//--------------------------------------------------------------------------------
// Stan maszyny naciśnieciu estopa 	
	E_Station.eAborting:                 	// Stan bezpiecznego zatrzymywania (po EStopie)
		bGate1:= FALSE;
		bGate2:= FALSE;
	
		ACT_ResetCommands();

		eState 						:=  E_Station.eAborted;  
		eRunningState				:=	E_CapFeederState.eReady;
		
//--------------------------------------------------------------------------------
// Stan masyzny po wykryciu błędu			
	E_Station.eError:                 	 	// Stan błędu 	
		
		ACT_ResetCommands();
		
		IF bReset THEN
			eState 				:= E_Station.eResetting;
			bError := FALSE;
		END_IF
		
//--------------------------------------------------------------------------------
// Stan masyzny po wykryciu błędu
	E_Station.eResetting:					// Stan resetowania bledu (po Errorze)
			CASE udiErrorID-udiStationIndex OF
		
				//Error 8 - Błąd falownika
				266:
					fbInverter.bReset	:= TRUE;
					bError 				:= FALSE;
				ELSE
					bError := FALSE;	
			END_CASE		
		
		IF NOT bError AND fbInverter.eState = E_Station.eReady THEN
			fbInverter.bReset	:= FALSE;	
			
			udiErrorID 			:=	0;
			sErrorDescription 	:=	'';
			eState 				:=	E_Station.ePreparingToReady;
			eRunningState		:=	E_CapFeederState.eReady;
		ELSE
			eState 				:=	E_Station.eError;
		END_IF
    
//--------------------------------------------------------------------------------
// Stan ruchoow manualnych
	E_Station.eManualMovement:     			// Stan ruchów manualnych  
   
		ACT_ManualMovements();
		//Wyjście z trybu serwisowego
		IF NOT bManualMovement THEN
			
			bHeightMotorUp				:=	FALSE;
			bHeightMotorDown			:=	FALSE;
			
			eState:=E_Station.eReady;
		END_IF
		

//--------------------------------------------------------------------------------
// Stan rozpoczecia bazowania
	E_Station.eHoming:						// Stan bazowania 
		
		ACT_Homing();
		IF NOT bHoming AND NOT bHeightSet THEN
			bHeightMotorDown					:=	FALSE;
			bHeightMotorUp						:=	FALSE;
		   eState								:=E_Station.ePreparingToReady;
		END_IF		
		
//--------------------------------------------------------------------------------
// Stan zakończenia bazowania
	E_Station.eHomingDone:                  // Stan wykonania bazowania 
	
		bHeightMotorDown					:=	FALSE;
		bHeightMotorUp						:=	FALSE;
		bHeightMotorEncoderCounterReset		:=	FALSE;
		bHomingDone							:=	TRUE;
		IF NOT bHoming AND NOT bHeightSet THEN
		   eState:=E_Station.eReady;
		END_IF
		
//--------------------------------------------------------------------------------
// Stan przygotowania do gotowości
	E_Station.ePreparingToReady:            // Stan przygotowywania do gotowosci (zawsze przed Ready)  
		
		bGate1:= FALSE;
		bGate2:= FALSE;
	
		bSorterEngine:=FALSE;
		bSorterAir:=FALSE;
		
		eRunningState:=E_CapFeederState.eReady;
		eState:=E_Station.eReady;	
		
//-------------------------------------------------------------------------------
// Stan przygotowania do wyłączenia maszyny
	E_Station.ePreparingToDisable:          // Stan przygotowywania do nieaktywnosci (po wyłączeniu Enable) 
		
		bGate1:= FALSE;
		bGate2:= FALSE;
	
		bSorterEngine:=FALSE;
		bSorterAir:=FALSE;
		bHeightMotorUp:= NOT tonHomingSensor.Q;
		bHeightMotorDown:=FALSE;	
		IF tonHeightNoChange.Q OR tonHeightNoChangeTime.Q THEN
			bHeightMotorUp			:=	FALSE;
			bHeightMotorDown		:=	FALSE;	
			eRunningState			:=	E_CapFeederState.eReady;		
			eState					:=	E_Station.eDisabled;
		END_IF	
			
//--------------------------------------------------------------------------------
// Stan gotowości
	E_Station.eReady:						// Stan gotowosci 
	
		IF bRun AND NOT bCycleDone AND NOT bCycleNotDone THEN
			eState 				:= E_Station.eStarting; 
		END_IF
		IF bHoming OR bHeightSet THEN
			bHomingDone							:=	FALSE;
			eState 								:= E_Station.eHoming; 
		END_IF
		IF bManualMovement THEN
			//Jeśli przejście w tryb ruchów manualnych przepisz wszystkie stany siłowników sterowanych przez moduł
			//aby zapobiec ewentualnym kolizjom po wejściu w tryb serwisowy
			
			bManualHeightMotorUp		:= bHeightMotorUp;
			bManualHeightMotorDown		:= bHeightMotorDown;
			
			eState 						:= E_Station.eManualMovement; 
		END_IF
		IF NOT bRun THEN
			bCycleDone 			:= FALSE;
			bCycleNotDone 		:= FALSE;			
		END_IF
		
//--------------------------------------------------------------------------------
// Stan zatrzymywania
	E_Station.eStopping:					// Stan zatrzymywania 
		
		bSorterAir 		:= 	TRUE;
		bSorterEngine 	:=	FALSE;
		IF tonStoppingTime.Q THEN
			ACT_ResetCommands();
			eRunningState							:= E_CapFeederState.eReady;
			eState									:= E_Station.eReady;
		END_IF

		
//--------------------------------------------------------------------------------
// Stan uruchomienia lini ( po eReady)
	E_Station.eStarting:                  	// Stan uruchamiania (po Ready)
		iValvesCycleCase		:=0;
		eState					 := E_Station.eRunning; 

//--------------------------------------------------------------------------------
// Stan wykonywania pracy
	E_Station.eRunning:               		// Stan wykonywania cyklu (po Startingu), w tym stanie osobny

		ACT_Running();
		IF NOT bRun THEN 					(*Przerywanie cyklu*)
			eState				:= E_Station.eStopping;
			//bCycleNotDone		:= TRUE;
		END_IF
		(*IF bCycleDone OR bCycleNotDone THEN (*Cykl zakończony*)
			eState 				 := E_Station.eReady;
		END_IF*)						
		
		
END_CASE
END_ACTION

ACTION ACT_ErrorHandling:
//OBSŁUGA BŁĘDÓW STACJI SPRAWDZANIA
//************LISTA BŁĘDÓW***************
bStateError:= (eState=E_Station.eError) OR (eState=E_Station.eResetting) OR bIgnoreError;

//************LISTA BŁĘDÓW***************

//Error 1 - podnośnik nie porusza się pomimo wysterowania 
tonErrorHeightChange(IN:=(bHeightMotorUp OR bHeightMotorDown) AND lrLastHeightMotorPositionCV=lrHeightMotorPositionCV, PT:=T#3S);
tonEmptySleeveError(IN:=NOT bFullSleeveSensor AND bRun, PT:=INT_TO_TIME(iTimeToEmptySleeveError)*1000); //Było 30, teraz jest z receptur
tonMaxHeightError(IN:=lrHeightMotorPositionSV>lrMaxHeight AND NOT bHomingNeeded AND eState=E_Station.eReady,PT:=T#30S);
tonMinHeightError(IN:=lrHeightMotorPositionSV<lrMinHeight AND NOT bHomingNeeded AND eState=E_Station.eReady,PT:=T#30S);
tonSorterEngineError(IN:= NOT bEngineOK AND bSorterEngine, PT:=T#3S);
tonInverterError(IN:=fbInverter.bError AND NOT bStateError, PT:=T#3S);

IF (bEnable OR (eState = E_Station.ePreparingToDisable)) AND NOT bIgnoreError THEN
	
	IF tonErrorHeightChange.Q THEN
		bError:=TRUE;
		udiErrorID:=261;
		//udiErrorID:= udiErrorID+udiStationIndex;
		sErrorDescription:='Blokada podnośnika lub brak zasilania - sprawdź czujnik lub odblokuj mechanicznie';	
		sErrorDescription2:='';
	END_IF
	
	
	IF tonSorterEngineError.Q THEN
		bError:=TRUE;
		udiErrorID:=262;
		//udiErrorID:= udiErrorID+udiStationIndex;
		sErrorDescription:='Bład zabezpieczenia silnika - sprawdź wyłącznik';	
		sErrorDescription2:='';	
	END_IF
	
	//Error 3 - Pusty rekaw sortera nasadek
	IF tonEmptySleeveError.Q THEN
		bError:=TRUE;
		udiErrorID:=263;
		//udiErrorID:= udiErrorID+udiStationIndex;
		sErrorDescription:='Pusty rękaw sortera - uzupełnij nasadki';
		sErrorDescription2:='';
	END_IF
	
	
	//Error 4 - Bład nastaw max
	IF tonMaxHeightError.Q  THEN
		bError:=TRUE;
		udiErrorID:=264;
		//udiErrorID:= udiErrorID+udiStationIndex;
		sErrorDescription:='Wartość zadana wysokości jest większa od maksymalnej - zmień ustawienia w recepturze';
		sErrorDescription2:=REAL_TO_STRING(LREAL_TO_INT(lrMaxHeight));
	END_IF
	
	//Error 5 - Bład nastaw min
	IF tonMinHeightError.Q THEN
		bError:=TRUE;
		udiErrorID:=265;
		//udiErrorID:= udiErrorID+udiStationIndex;
		sErrorDescription:='Wartość zadana wysokości jest mniejsza od minimalnej - zmień ustawienia w recepturze ';
		sErrorDescription2:=REAL_TO_STRING(LREAL_TO_INT(lrMinHeight));
	END_IF	
	
	//Error 6 - Bład falownika
	IF tonInverterError.Q THEN
		bError:=TRUE;
		udiErrorID:=266;
		//udiErrorID:= udiErrorID+udiStationIndex;
		sErrorDescription:='Błąd falownika';
		sErrorDescription2:='';
	END_IF		
	
	
	
ELSE
	bError	:=FALSE;
END_IF


//-----------------------------------------------------------------------
IF bError AND NOT bStateError THEN

	IF eLastState = eRunning THEN
		bCycleNotDone						:= TRUE;
	END_IF

	eState 									:= E_Station.eError;
END_IF


//------------------------------------------------------------------------

(*Wyświetlanie błedu na wyjściu*)
bError;

(*Przepisywanie nazwy stacji*)
sErrorStationName 							:= sStationName;

//Jezeli nie zbazowane to potrzebne bazowanie
IF NOT bHeightMotorEncoderHomed  THEN
	bHomingDone								:=	FALSE;
END_IF
END_ACTION

ACTION ACT_HeightMotor:
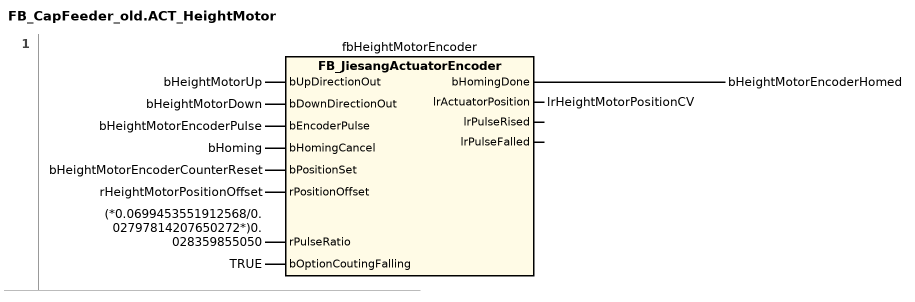
// NETWORK 1
fbHeightMotorEncoder(
    bUpDirectionOut := bHeightMotorUp,
    bDownDirectionOut := bHeightMotorDown,
    bEncoderPulse := bHeightMotorEncoderPulse,
    bHomingCancel := bHoming,
    bPositionSet := bHeightMotorEncoderCounterReset,
    rPositionOffset := rHeightMotorPositionOffset,
    rPulseRatio := (*0.0699453551912568/0.02797814207650272*)0.028359855050,
    bOptionCoutingFalling := TRUE,
    lrActuatorPosition => lrHeightMotorPositionCV); // FB_JiesangActuatorEncoder
bHeightMotorEncoderHomed := fbHeightMotorEncoder.bHomingDone;
END_ACTION

ACTION ACT_Homing:
//BAZOWANIE

tofHeightMotorDown(IN:=bHeightMotorDown, PT:=T#1S); //Zabezpieczenie przed zbyt szybkim przełączeniem pomiędzy Down a Up, bezpiecznieki sie palą
	
//Podnoszenie stacji do maksymalnej pozycji
IF NOT bHeightMotorEncoderHomed OR rtEncoderHomed.Q THEN
	bHeightMotorUp:=(*TRUE*) NOT tofHeightMotorDown.Q AND NOT tonHomingSensor.Q;
	bHeightMotorDown:=FALSE;
	IF tonHeightNoChange.Q OR tonHeightNoChangeTime.Q THEN
		bHeightMotorEncoderCounterReset:=TRUE;
		bHeightMotorUp:=FALSE;
    END_IF
	//Jesli enkoder zbazowany zakończ bazowanie	
	IF rtEncoderHomed.Q  THEN
		bHeightMotorUp:=FALSE;
		bHeightMotorDown:=FALSE;
		eState:=E_Station.eHomingDone;
	END_IF		
		
//Po podniesieniu stacji opuszczanie do ustalonej wysokości
ELSIF bHeightMotorEncoderHomed THEN
	bHeightMotorEncoderCounterReset:=FALSE;
	bHeightMotorUp:=lrHeightMotorPositionCV<=lrHeightMotorPositionSV;
	bHeightMotorDown:=lrHeightMotorPositionCV>=lrHeightMotorPositionSV;
	//Kiedy stacja osiągnie wysokość zadaną
	IF ABS(lrHeightMotorPositionCV-lrHeightMotorPositionSV)<0.5 OR tonLimitPosMaxReachedDelay.Q OR tonLimitPosMinReachedDelay.Q THEN
		bHeightMotorDown:=FALSE;
		bHeightMotorUp:=FALSE;
		eState:=E_Station.eHomingDone;
	END_IF			
END_IF
END_ACTION

ACTION ACT_Inverter:
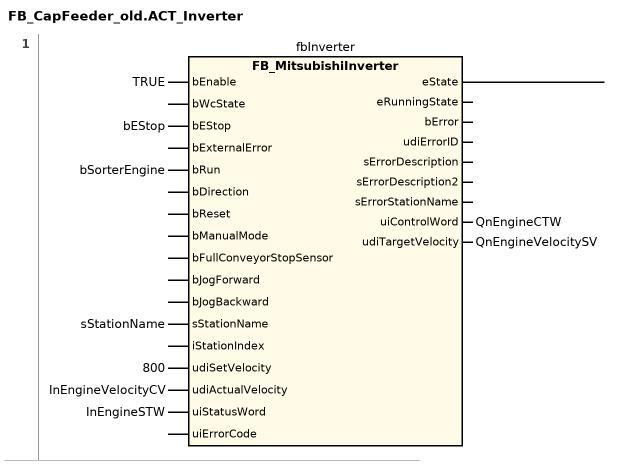
// NETWORK 1
fbInverter(
    bEnable := TRUE,
    bEStop := bEStop,
    bRun := bSorterEngine,
    sStationName := sStationName,
    udiSetVelocity := 800,
    udiActualVelocity := InEngineVelocityCV,
    uiStatusWord := InEngineSTW,
    uiControlWord => QnEngineCTW,
    udiTargetVelocity => QnEngineVelocitySV); // FB_MitsubishiInverter
END_ACTION

ACTION ACT_Limits:
IF iTimeToEmptySleeveError < 5 THEN
	iTimeToEmptySleeveError := 5;
END_IF
END_ACTION

ACTION ACT_ManualMovements:
//W trybie ruchów manualnych wykonuj ruchy za pomocą rozkazów manualnych
IF NOT bRun THEN
	
	bHeightMotorUp:=bManualHeightMotorUp;
	bHeightMotorDown:=bManualHeightMotorDown;
	bSorterEngine:=bManualSorterEngine;
	bSorterAir:=bManualSorterAir;
	
	bGate1:=bManualGate1; //Not dla tego, że defoltowy stan WYSUNIĘTY (true)
	bGate2:=bManualGate2; //Not dla tego, że defoltowy stan WYSUNIĘTY (true)

(*ELSE	//Kasuje zeby po cyklu nic sie nie poruszało

	bManualHeightMotorUp 	:= FALSE;
	bManualHeightMotorDown  := FALSE;
	bSorterEngine	:=FALSE;
	bSorterAir		:=FALSE;
*)	
END_IF


IF bHoming OR bHeightSet THEN
	eState:=E_Station.eHoming;
END_IF

IF bRun THEN	
	ACT_Running();
END_IF
//Zabezpieczenie przed kolizją stacji poprzez ruch podnośnika	
IF bHeightMotorDown AND lrHeightMotorPositionCV<=lrMinHeight AND NOT bHoming AND NOT bHeightSet THEN
	bHeightMotorDown:=FALSE;
END_IF	

IF bHeightMotorUp AND lrHeightMotorPositionCV>=lrMaxHeight AND NOT bHoming AND NOT bHeightSet THEN
	bHeightMotorUp:=FALSE;
END_IF
END_ACTION

ACTION ACT_ResetCommands:
//Reset komend ruchu 	


bHeightMotorUp				:=	FALSE;
bHeightMotorDown			:=	FALSE;
bSorterAir 		:= 	FALSE;
bSorterEngine 		:=	FALSE;
END_ACTION

ACTION ACT_Running:
//----------------------------------------------------------------------------------
// Obsługa podajnik zamknięc


(*CASE iValvesCycleCase OF
	0:
		bGate1:= FALSE;
		IF (tonGates1.Q) THEN
			iValvesCycleCase :=1;
		END_IF
	1:
		bGate1:= TRUE;
		IF (tonGates2.Q) THEN
			iValvesCycleCase :=2;
		END_IF	
	2:
		bGate2:= FALSE;
		IF (tonGates3.Q) THEN
			iValvesCycleCase :=3;
		END_IF
	3:
		bGate2:= TRUE;
		IF (tonGates4.Q) THEN
			iValvesCycleCase :=0;
		END_IF	
END_CASE*)

//rtOutSensor(CLK:=P08_CapSorter.IbCapSorterGateGateAfterSensor);
	
CASE iValvesCycleCase OF
	0:
		//IF (rtOutSensor.Q) THEN
		IF (NOT bSensorInPipe) THEN

			iValvesCycleCase:=1;
		END_IF
		;
	1:
		bGate1:= TRUE;
		IF (tonGates1.Q) THEN
			iValvesCycleCase :=2;
		END_IF
	2:
		bGate1:= FALSE;
		IF (tonGates2.Q) THEN
			iValvesCycleCase :=3;
		END_IF	
	3:
		bGate2:= TRUE;
		IF (tonGates3.Q) THEN
			iValvesCycleCase :=4;
		END_IF
	4:
		bGate2:= FALSE;
		IF (tonGates4.Q) THEN
			iValvesCycleCase :=0;
		END_IF	
END_CASE

CASE eRunningState OF
	
	//NIEGOTOWY
	E_CapFeederState.eDisabled:
		eRunningState:=E_CapFeederState.eReady;

	E_CapFeederState.eReady:
		iTryUnblockWheel		:=	0;
		bTryUnblockWheel		:= FALSE;	
		fbInverter.bDirection 	:= FALSE;
		IF bRun THEN
			eRunningState			:=E_CapFeederState.eSorting;
		END_IF
	
	
	E_CapFeederState.eSorting:
	
		bSorterEngine:=tonAirBeforeStart.Q;
		bSorterAir:=(	//Nie wiem co to za wymysły
						(aBufferedSensorValue[20](*tofCapFeederSorterCapSensor.Q*) OR NOT tonAirBeforeStart2.Q)(* AND bImpON*)AND NOT bBlowDelay
					)	OR	
					bTryUnblockWheel // Dmuchanie jeżeli jest obrót do tyłu
;
		//aBufferedSensorValue[20] - 20 to jest opóznenie (buferizacja signala czujnika w cyklach programy (3ms x 20 = 60 ms). Czas opóznenia 
		//możemy obliczyć od prędcosci falownika i prszykładni: mamy 51 gniazdk0, 800 rpm, przykladnia 1:40 => mamy 800/40=20rmp, /60 =>
		//0,33 obrota / sec => 0,33 obrota/sec * 51 dnazdko/obrot = 17 gniazdek/sek => 1/17 = 0,059sec/1gniazdko => opoznenie 60 ms
		//60ms/3ms(czas cyclu) => 20 cyclów
		
		(*Próba odblokowania koła*)
			iTryUnblockWheel := iTryUnblockWheel + 1;
			IF rtCapSorterSensor.Q THEN
				iTryUnblockWheel	:=	0;
			END_IF
			IF tonEngineBlocked.Q THEN
				bTryUnblockWheel := TRUE;
			END_IF	
			IF bTryUnblockWheel THEN
				fbInverter.bDirection := TRUE;
			END_IF
			IF tonTryUnblockWheel.Q THEN
				iTryUnblockWheel		:=	0;//dp
				bTryUnblockWheel		:= FALSE;
				fbInverter.bDirection 	:= FALSE;
			END_IF
		(* Koniec Próba odblokowania koła*)	
		
		IF tonSortingEngineOff.Q THEN 
			eRunningState 			:=E_CapFeederState.eSleeveFull;
		END_IF
	
	E_CapFeederState.eSleeveFull:
	
		bSorterEngine:=FALSE;
		bSorterAir:=NOT tonAirAfterStop.Q(* AND bImpON*);
		IF tonAirAfterStop.Q THEN
			IF tonSortingEngineOn.Q THEN
				eRunningState		:=E_CapFeederState.eSorting; 
			END_IF
		END_IF
	
	E_CapFeederState.eSleeveLowLevel:
	
			//Wlaczenie silnika i zaworu po czasie
		bSorterEngine:=TRUE;
		bSorterAir:=tofCapFeederSorterCapSensor.Q (*AND bImpON*);
		IF tonSortingEngineOff.Q THEN
			eRunningState		 	:=E_CapFeederState.eSorting;
		END_IF
	
END_CASE
END_ACTION

ACTION ACT_Signals:
(** Timery na potrzeby bazowania**)
rtEncoderHomed(CLK:=bHeightMotorEncoderHomed,Q=>);
tonHeightNoChange(IN:=((bHeightMotorUp OR bHeightMotorDown OR tonHomingSensor.Q) AND (lrLastHeightMotorPositionCV=lrHeightMotorPositionCV)), PT:=T#500MS); 
tonHomingSensor(IN:=(bHomingSensor), PT:=T#100MS);
//tonHeightNoChangeTime(IN:=(eState = E_Station.eHoming OR eState = E_Station.ePreparingToDisable) AND bHeightMotorUp, PT:=T#8S); 

tonLimitPosMinReachedDelay(IN:=(lrHeightMotorPositionCV<=lrMinHeight) AND eState=E_Station.eHoming,PT:=T#2S);
tonLimitPosMaxReachedDelay(IN:=(lrHeightMotorPositionCV>=lrMaxHeight) AND eState=E_Station.eHoming,PT:=T#2S);
	
(** Timery używane podczas pracy stacji**)
tonSortingEngineOff(IN:=((eRunningState=E_CapFeederState.eSorting OR eRunningState=E_CapFeederState.eSleeveLowLevel) AND bRun AND bFullSleeveSensor),PT:=INT_TO_TIME(iTimeDelayOff));
tonSortingEngineOn(IN:=((eRunningState=E_CapFeederState.eSorting OR eRunningState=E_CapFeederState.eSleeveFull) AND bRun AND NOT bFullSleeveSensor),PT:=INT_TO_TIME(iTimeDelayOn));
tonSleeveFullEngineOn(IN:=(eRunningState=E_CapFeederState.eSleeveFull AND bRun AND NOT bFullSleeveSensor),PT:=INT_TO_TIME(iTimeDelayOff));
rtCapSorterSensor(CLK:=bSorterCapSensor, Q=>);
tonEngineBlocked(IN:=iTryUnblockWheel > 1500 AND bSorterEngine AND NOT bTryUnblockWheel,PT:=T#1MS); //Zablokowany silnik
tonTryUnblockWheel(IN:=bTryUnblockWheel, PT:=T#1S900MS);
tofCapFeederSorterCapSensor(IN:=tonCapFeederSorterCapSensor.Q,PT:=T#10MS); //bylo 200
tonCapFeederSorterCapSensor(IN:=bSorterCapSensor,PT:=T#3mS);//było 3ms
tonAirBeforeStart(IN:=eRunningState=E_CapFeederState.eSorting, PT:=T#1S);
rtCapFeederSorterCapSensor(CLK:=tofCapFeederSorterCapSensor.Q,Q=>);

tonAirBeforeStart2(IN:=eRunningState=E_CapFeederState.eSorting, PT:=T#2S);
tonAirAfterStop(IN:=eRunningState=E_CapFeederState.eSleeveFull, PT:=T#2S);

//prszesunęcie wartosci czujnika po buforu opoznenia 

FOR i:=40 TO 1 BY -1 DO
	aBufferedSensorValue[i] := aBufferedSensorValue[i-1];
END_FOR
aBufferedSensorValue[0] := bSorterCapSensor;

IF rtCapFeederSorterCapSensor.Q THEN
	bBlowDelay := TRUE;
	
END_IF
tonbBlowDelay(IN:=bBlowDelay,PT:=T#35MS);
IF tonbBlowDelay.Q THEN
	bBlowDelay:= FALSE;
END_IF
TimerOn (IN := NOT bImpOn, PT := T#10MS);
IF TimerOn.Q THEN
	bImpOn := TRUE;
END_IF
TimerOff (IN := bImpOn, PT := T#10MS);
IF TimerOff.Q THEN
	bImpON := FALSE;
END_IF

//Czasówki pneumatiki
//tonGates1(IN:= (iValvesCycleCase = 0 AND (eState = E_Station.eRunning OR eState = E_Station.eManualMovement)), PT:=T#300MS);//150//300
//tonGates2(IN:= (iValvesCycleCase = 1 AND (eState = E_Station.eRunning OR eState = E_Station.eManualMovement)), PT:=T#200MS);//500//300
//tonGates3(IN:= (iValvesCycleCase = 2 AND (eState = E_Station.eRunning OR eState = E_Station.eManualMovement)), PT:=T#300MS);//150//300
//tonGates4(IN:= (iValvesCycleCase = 3 AND (eState = E_Station.eRunning OR eState = E_Station.eManualMovement)), PT:=T#200MS);//500//300

//Czasówki pneumatiki
tonGates1(IN:= (iValvesCycleCase = 1 AND (eState = E_Station.eRunning OR eState = E_Station.eManualMovement)), PT:=T#200MS);//150//300
tonGates2(IN:= (iValvesCycleCase = 2 AND (eState = E_Station.eRunning OR eState = E_Station.eManualMovement)), PT:=T#200MS);//500//300
tonGates3(IN:= (iValvesCycleCase = 3 AND (eState = E_Station.eRunning OR eState = E_Station.eManualMovement)), PT:=T#200MS);//150//300
tonGates4(IN:= (iValvesCycleCase = 4 AND (eState = E_Station.eRunning OR eState = E_Station.eManualMovement)), PT:=T#200MS);//500//300


(** Dodatkowy timer przy zatrzymywaniu**)
tonStoppingTime( IN:= eState= E_Station.eStopping, PT:=T#2S);
END_ACTION

ACTION ACT_Statistic:
//Statystyka do zliczania czasu cyklu 
rtrigCycleTimerRead(CLK:=eRunningState=E_CapFeederState.eSleeveFull OR eRunningState=E_CapFeederState.eSleeveLowLevel);

	IF rtrigCycleTimerRead.Q THEN
		tCycleTime:=tonCycleTimer.ET;
		
	END_IF
	
tonCycleTimer(IN:=eRunningState= E_CapFeederState.eSorting , PT:=T#1D);
END_ACTION

ACTION ACT_Status:

(*Zapisywanie ostatniego stanu*)
	IF eLastStateTemp<>eState THEN
		eLastState := eLastStateTemp;
	END_IF
	eLastStateTemp := eState;
	
	IF eLastRunningStateTemp<>eRunningState THEN
		eLastRunningState := eLastRunningStateTemp;
	END_IF
	eLastRunningStateTemp := eRunningState;
(*Koniec Zapisywanie ostatniego stanu*)
END_ACTION

ACTION ACT_Warnings:
//Usrawianie warningów

//Filtrowanie czujnika ultradźwiękowego
fbbLevelSensor	(bIN:=NOT bLevelSensor AND (eRunningState=E_CapFeederState.eSorting OR eRunningState=E_CapFeederState.eSleeveLowLevel OR eRunningState=E_CapFeederState.eSleeveFull) , tFilterTimeOn:= T#5S, tFilterTimeOff:=T#5S , bOUT=> );


IF fbbLevelSensor.bOUT THEN
		bWarning1						:=	TRUE;			
		udiWarningID					:=	1;
		sWarningDescription				:=	'Nieski poziom w sorterze nasadek';
ELSE
		bWarning1						:=	FALSE;			
		udiWarningID					:=	0;
		sWarningDescription				:=	'';
END_IF
END_ACTION

ACTION aStationID:
udiStationID	:=	udiStationIndex;
END_ACTION

END_FUNCTION_BLOCK

// ---- POUs/FB/FB_CatchStationEnkoder.TcPOU
(*
Nazwa:			FB_CatchStation
Opis:			Chwytak pod stacjami 
Wersja:			v1.1
Data:			2023-02-22
Autor:			TW,DP
Urzadzenia:		Silownik chwytania, podnośnik JIESANG
Konfiguracja:	
Zmiany:
20230222 - Zwieksozmny czas bledu 9
Info:
- dodano błędy od nastaw powyżej max i min (error 7 i 8)
- dodawno bHomingNeeded
- wylaczanie wyjść zmiana 2 wylaczanie wyjsc jak zniknie Enable
*)


FUNCTION_BLOCK FB_CatchStationEnkoder
VAR_INPUT
	bEnable: BOOL;						//Zezwolenie na pracę
	bEStop:BOOL;						//Stop Awaryjny włączony
	bRun:BOOL;							//Rozkaz łapania 
	bHoming:BOOL;						//Zezwolenie na wykonanie bazowania i pozycjonowania podajnika
	bHeightSet:BOOL;					//Ustaw wysokość
	bChangeover:BOOL;					//Ustawianie na zadaną wysokość do wymiany elementów formatowych
	bChangeOver2:BOOL;
	bIgnoreError:BOOL;					//Ignorowania błędów cyklu pracy
	bReset:BOOL;						//Reset błędu, jeśli w stanie "eError"
	nGripperScrewerPosition   	:LREAL; // Aktualna pozycja serwa od podnoszenia
	nSafetyScrewerPosition		:LREAL;	// zadana bezpieczna pozycja 
	bScrewerbError				:BOOL;  // Sygnał błędu od zakręcarki
	nPositionHeightSV:LREAL;			//Wysokość zadana na której ma znajdować się stacja
	bOpenedActuatorSensor:BOOL;			//Czujnik otwarcia siłownika łapania
	bClosedActuatorSensor:BOOL;			//Czujnik otwarcia siłownika łapania
	lrMaxHeight:LREAL;					//Maksymalna wysokość podnośnika chwytaka
	lrMinHeight:LREAL;					//Minimalna wysokość podnośnika chwytaka
	bManualMovement:BOOL;				//Zezwolenie na ruchy ręcznę
	bUnlockColision:BOOL:=FALSE;		//Odblokowywanie możliwośći kolizji
	bAlarmSVCVDiffHeightDisable:BOOL;	//Wyłączenie alarmu od rożnicy wysokości zadanej od aktualnej
	bNoLifter:BOOL;						//Podnośnik
	
	_HEIGHTMOTOR_ 				:BOOL;
	udiHeightMotorEncoderVal	:UDINT;		//Ilość impulsów z modułu enkoderowego
	bHeightEncoderSetValDone	:BOOL;		//Zerowanie enkodera wykonane
	bHeightMotorEncoderPulse 	:BOOL;			//Sygnał impulsów enkodera siłownika
	rHeightMotorPositionOffset 	:REAL;		//Wysokość bazowani podnośnika

	_ALARMINFO_ :BOOL;
	iStationIndex:UDINT;					//Numer stacji 
	sStationName:STRING;					//Nazwa stacji	

	
END_VAR
VAR_OUTPUT
	eState: E_Station;						//Stan ogólny bloku
	eRunningState: E_CatchStationState;		//Stan wewnętrzny
	bError: BOOL;							//Błąd stacji
	nErrorNr: UDINT;						//Nr błędu podajnika platynek
	sErrorDescription:STRING(200);				//Opis błędu
	sErrorDescription2: STRING(200);				//Opis błędu 2
	sErrorStationName:STRING;				//Nazwa stacji
	udiStationID: UDINT;				// Nr stacji

	bCatchActuator:BOOL;					//Sterownie siłownika łapania opakowania
	bHeightMotorUp:BOOL;					//Sterowanie silnikiem podnośnika  - RUCH W GÓRĘ
	bHeightMotorDown:BOOL;					//Sterowanie silnikiem podnośnika  - RUCH W DÓŁ
	udiHeightMotorEncoderSetVal	:UDINT;		
	bHeightEncoderSetVal	:BOOL;		//Zerowanie enkodera
	lrHeightMotorCV:LREAL;					//Aktualna pozycja podnośnika
	tCycleTime:TIME;
	bHomingDone:BOOL;						//Wymagane ponowne bazowanie (blad podczas bazowania lub stop awaryjny)
	bCycleDone:BOOL;
	bCycleNotDone:BOOL;
END_VAR
VAR
	tonHeightNoChange: TON; 			//Timer wykrycia braku ruchu siłownika zmiany wysokości stacji
	nLastPositionHeightCV: LREAL;		//Pozycja podnośnika w poprzednim cyklu programu
	tonErrorHeightChange: TON; 			//Timer błędu podnośnika
	// Czas zadziałania siłownika
	tonCatchingTime: TON;
	// Timer blokady otwierania chwytaka
	tonOpeningBlocked: TON;
	rtEncoderHomed:R_TRIG;
	tonCycleTimer:TON;
	rtrigCycleTimerRead:R_TRIG;
	
	tofMotorUpPermition: TOF;
	tofMotorDownPermition: TOF;
	tonLimitPosMinReachedDelay: TON;
	tonLimitPosMaxReachedDelay: TON;
	tonMaxHeight		: TON;
	tonMinHeight		: TON;
	tonSVCVDiffHeight	: TON;
	
	//Podnośnik Jiesang	
	fbHeightMotorEncoder: FB_JiesangActuatorEncoderModul;//FB_JiesangActuatorEncoder;	// Blok enkodera podnośnika chwytaka stabilizującego pod zakręcarką	
	bHeightMotorEncoderCounterReset:BOOL; 				//Sygnał resetu enkodera
	bHeightMotorEncoderHomed:BOOL;						//Informacja od enkodera że jest zbazowany

	eLastState: E_Station;							//Stan ogólny bloku
	eLastRunningState: E_CatchStationState;			//Stan podbloku
	eLastStateTemp: E_Station;						//Stan ogólny bloku
	eLastRunningStateTemp: E_CatchStationState;		//Stan podbloku
	bStateError: BOOL;

	tonStopping: TON;
	tofHeightMotorDown: TOF;
	iCaseChangeover: INT;
	tonChangeOverLimitPosMinReachedDelay: TON;
	tonChangeoverLimitPosMaxReachedDelay: TON;
END_VAR

VAR_IN_OUT
	bManualCatchActuator:BOOL;		//Ruch ręczny siłownikiem podajnika platynek
	bManualHeightMotorUp:BOOL;			//Ruch ręczny podnośnika stacji w górę
	bManualHeightMotorDown:BOOL;		//Ruch ręczny podnośnika stacji w dół
END_VAR

HeightMotor();
ErrorHandling();
Control();
Changeover();
Statistics();
aStationID();
(*Zapisywanie ostatniego stanu*)
IF eLastStateTemp<>eState THEN
	eLastState := eLastStateTemp;
END_IF
eLastStateTemp := eState;
IF eLastRunningStateTemp<>eRunningState THEN
	eLastRunningState := eLastRunningStateTemp;
END_IF
eLastRunningStateTemp := eRunningState;
(*Koniec Zapisywanie ostatniego stanu*)


nLastPositionHeightCV:=lrHeightMotorCV;

ACTION aStationID:
udiStationID	:=	iStationIndex;
END_ACTION

ACTION Changeover:
tonChangeOverLimitPosMinReachedDelay(IN:=(lrHeightMotorCV<=lrMinHeight) AND bChangeover,PT:=T#2S);
tonChangeoverLimitPosMaxReachedDelay(IN:=(lrHeightMotorCV>=lrMaxHeight) AND bChangeover,PT:=T#2S);


//Przeniesione do PreparingToDisabled
(*CASE iCaseChangeover OF
	
	0: //Włączenie ustawiania
		IF bChangeover THEN
			iCaseChangeover := iCaseChangeover + 10;
			bHeightMotorDown:=FALSE;
			bHeightMotorUp:=FALSE;
		END_IF
		
	10: //Ustawianie stacji na wysokość 
		IF bHeightMotorEncoderHomed THEN
			bHeightMotorEncoderCounterReset	:=	FALSE;
			bHeightMotorUp					:=	lrHeightMotorCV	<=	200;
			bHeightMotorDown				:=	lrHeightMotorCV	>=	200;
			//Kiedy stacja osiągnie wysokość zadaną
			IF ABS(lrHeightMotorCV-nPositionHeightSV)<2 OR tonChangeoverLimitPosMaxReachedDelay.Q OR tonChangeOverLimitPosMinReachedDelay.Q  THEN
				bHeightMotorDown			:=	FALSE;
				bHeightMotorUp				:=	FALSE;
				iCaseChangeover 			:=	iCaseChangeover + 10;
			END_IF			
		ELSE
			bHeightMotorDown		:=	FALSE;
			bHeightMotorUp			:=	FALSE;
			iCaseChangeover 		:=  0;
		END_IF	
		
	20: //Czekanie na wyłączenie przezbrajania i ustawienie na odpowiednią wysokość z receptury
			IF NOT bChangeover THEN
				iCaseChangeover := iCaseChangeover + 10;
			END_IF
	30: //Ustawianie stacji na wysokość z receptury
		IF bHeightMotorEncoderHomed THEN
			bHeightMotorEncoderCounterReset	:=	FALSE;
			bHeightMotorUp					:=	lrHeightMotorCV	<=	nPositionHeightSV;
			bHeightMotorDown				:=	lrHeightMotorCV	>=	nPositionHeightSV;
			//Kiedy stacja osiągnie wysokość zadaną
			IF ABS(lrHeightMotorCV-nPositionHeightSV)<2 OR tonChangeoverLimitPosMaxReachedDelay.Q OR tonChangeOverLimitPosMinReachedDelay.Q  THEN
				bHeightMotorDown			:=	FALSE;
				bHeightMotorUp				:=	FALSE;
				iCaseChangeover 			:=	iCaseChangeover + 10;
			END_IF			
		ELSE
			bHeightMotorDown		:=	FALSE;
			bHeightMotorUp			:=	FALSE;
			iCaseChangeover 		:=  0;
		END_IF
	40: //Ustawianie stacji na wysokość z receptury	
		iCaseChangeover 		:=  0;

END_CASE
*)
END_ACTION

ACTION Control:

	(** TIMERY**)
	rtEncoderHomed(CLK:=bHeightMotorEncoderHomed,Q=>);
	tonHeightNoChange(IN:=((bHeightMotorUp OR bHeightMotorDown) AND (nLastPositionHeightCV=lrHeightMotorCV)), PT:=T#1S); 
	tonLimitPosMinReachedDelay(IN:=(lrHeightMotorCV<=lrMinHeight) AND eState=E_Station.eHoming,PT:=T#2S);
	tonLimitPosMaxReachedDelay(IN:=(lrHeightMotorCV>=lrMaxHeight) AND eState=E_Station.eHoming,PT:=T#2S);
	tonStopping(IN:=eState=E_Station.eStopping,PT:=T#2S);
	tofMotorUpPermition(IN:=bHeightMotorDown,PT:=T#250MS);
	tofMotorDownPermition(IN:=bHeightMotorUp ,PT:=T#250MS);	
	(*****Wyłączenie enable*****)
	IF NOT bEnable OR bChangeover THEN //Lub przezbrajania
		IF eState <> E_Station.eDisabled AND eState <> E_Station.ePreparingToDisable AND nGripperScrewerPosition>nSafetyScrewerPosition AND NOT bScrewerbError THEN
				eState 				:= E_Station.ePreparingToDisable; 
		END_IF	
	END_IF

	(*****Estop*****)
	IF NOT bEstop  THEN	
		IF eState <> E_Station.eAborted AND eState <> E_Station.eAborting AND eState <> E_Station.eDisabled THEN
				eState 				:= E_Station.eAborting; 
		END_IF
	END_IF

	CASE eState OF
	/////////////////////////////	
		E_Station.eDisabled: 					// Stan nieaktywnosci (Stacja wyłączona) 

			IF bEnable THEN
				eState 				:= E_Station.ePreparingToReady; 
			END_IF 
			
    /////////////////////////////	    
		E_Station.eAborted: 					// Stan bezpiecznego zatrzymania (po Abortingu) 

			IF bEStop THEN
				eState 				:= E_Station.ePreparingToReady;
			END_IF
			
	/////////////////////////////	
		E_Station.eAborting:                 	// Stan bezpiecznego zatrzymywania (po EStopie)

			bHeightMotorUp				:=	FALSE;
			bHeightMotorDown			:=	FALSE;
			eState := E_Station.eAborted;  
			eRunningState:=E_CatchStationState.eDisabled;
			
	/////////////////////////////			
		E_Station.eError:                 	 	// Stan błędu 	

			iCaseChangeover 		:=	0;
			IF bReset THEN
				eState 				:=	E_Station.eResetting;
			END_IF
						
	/////////////////////////////
		E_Station.eResetting:					// Stan resetowania bledu (po Errorze)
	
			bError := FALSE;

			IF NOT bError THEN
				nErrorNr 			:=	0;
   				sErrorDescription 	:=	'';
				eState 				:=	E_Station.ePreparingToReady;
			ELSE
				eState 				:=	E_Station.eError;
			END_IF
        
	/////////////////////////////
		E_Station.eManualMovement:     			// Stan ruchów manualnych  

			ManualMovements();
			//Wyjście z trybu serwisowego
			IF NOT bManualMovement THEN
				bCatchActuator				:=	FALSE;
				bHeightMotorUp				:=	FALSE;
				bHeightMotorDown			:=	FALSE;
				bManualCatchActuator		:=	bCatchActuator;
				eState:=E_Station.eReady;
			END_IF

	/////////////////////////////
		E_Station.eHoming:						// Stan bazowania 
	IF (nGripperScrewerPosition>nSafetyScrewerPosition AND NOT bScrewerbError) OR bManualMovement THEN  // co to za bzdura
			Homing();
			IF NOT bHoming AND NOT bHeightSet THEN // co to za bzdura
			   eState:=E_Station.ePreparingToReady;
			   	bHeightMotorDown:=FALSE;
				bHeightMotorUp:=FALSE;
			END_IF		
	END_IF		
	/////////////////////////////
		E_Station.eHomingDone:                  // Stan wykonania bazowania 
	
			bHeightMotorDown					:=	FALSE;
			bHeightMotorUp						:=	FALSE;
			bHeightMotorEncoderCounterReset		:=	FALSE;
			bHomingDone							:=	TRUE;
			IF NOT bHoming AND NOT bHeightSet THEN
			   eState:=E_Station.eReady;
			END_IF
			
	/////////////////////////////
		E_Station.ePreparingToReady:            // Stan przygotowywania do gotowosci (zawsze przed Ready)  
	
			bCatchActuator	:=	FALSE;
			eRunningState	:=	E_CatchStationState.eReady;
			eState			:=	E_Station.eReady;	
			
	/////////////////////////////
		E_Station.ePreparingToDisable:          // Stan przygotowywania do nieaktywnosci (po wyłączeniu Enable) 
  
			bCatchActuator:=FALSE;
			IF NOT bChangeOver THEN //Normalne wyłączenie
				bHeightMotorUp:=TRUE;
				bHeightMotorDown:=FALSE;	
				IF tonHeightNoChange.Q THEN
					bHeightMotorUp:=FALSE;
					eState:=E_Station.eDisabled;
					eRunningState:=E_CatchStationState.eDisabled;
				END_IF	
			ELSE //Wyłączenie z przebrajaniem na pozycje 200
				IF bHeightMotorEncoderHomed THEN
					bHeightMotorEncoderCounterReset	:=	FALSE;
					bHeightMotorUp					:=	lrHeightMotorCV	<=	150 AND NOT tofMotorUpPermition.Q;
					bHeightMotorDown				:=	lrHeightMotorCV	>=	150 AND NOT tofMotorDownPermition.Q;
					//Kiedy stacja osiągnie wysokość zadaną
					IF ABS(lrHeightMotorCV-150)<2 OR tonChangeoverLimitPosMaxReachedDelay.Q OR tonChangeOverLimitPosMinReachedDelay.Q  THEN
						bHeightMotorDown			:=	FALSE;
						bHeightMotorUp				:=	FALSE;
						eState						:=	E_Station.eDisabled;
						eRunningState				:=	E_CatchStationState.eDisabled;
					END_IF			
				ELSE
					bHeightMotorDown				:=	FALSE;
					bHeightMotorUp					:=	FALSE;
					eState								:=E_Station.eDisabled;
					eRunningState					:=	E_CatchStationState.eDisabled;
				END_IF	
			END_IF
				
	/////////////////////////////
		E_Station.eReady:						// Stan gotowosci 

			IF bRun AND NOT bCycleDone AND NOT bCycleNotDone THEN
				eState 				:= E_Station.eStarting; 
			END_IF
			IF bHoming OR bHeightSet OR bChangeover THEN
				eState 				:= E_Station.eHoming; 
			END_IF
			IF bManualMovement THEN
				//Jeśli przejście w tryb ruchów manualnych przepisz wszystkie stany siłowników sterowanych przez moduł
				//aby zapobiec ewentualnym kolizjom po wejściu w tryb serwisowy
				bManualCatchActuator		:= bCatchActuator;
				bManualHeightMotorUp		:= bHeightMotorUp;
				bManualHeightMotorDown		:= bHeightMotorDown;
				
				eState 						:= E_Station.eManualMovement; 
				eRunningState 				:= E_CatchStationState.eReady;
 
			END_IF
			IF NOT bRun THEN
				bCycleDone 			:= FALSE;
				bCycleNotDone 		:= FALSE;			
			END_IF
			
	/////////////////////////////
		E_Station.eStopping:					// Stan zatrzymywania 
					
			Running();
			IF bOpenedActuatorSensor OR tonStopping.Q THEN //NEW
				eState						:=	E_Station.eReady;
				eRunningState 				:=	E_CatchStationState.eReady;
			END_IF
			
	/////////////////////////////
		E_Station.eStarting:                  	// Stan uruchamiania (po Ready)
				
			eState					 := E_Station.eRunning; 

	/////////////////////////////
		E_Station.eRunning:               		// Stan wykonywania cyklu (po Startingu), w tym stanie osobny

			Running();
			IF NOT bRun THEN 					(*Przerywanie cyklu*)
				eState				:= E_Station.eStopping;
				bCycleNotDone		:= TRUE;
			END_IF
			(*IF bCycleDone OR bCycleNotDone THEN (*Cykl zakończony*)
				eState 				 := E_Station.eReady;
			END_IF*)						
		ELSE
		
		
	/////////////////////////////		
	END_CASE
END_ACTION

ACTION ErrorHandling:
//OBSŁUGA BŁĘDÓW PODAJNIKA PLATYNEK

//************LISTA BŁĘDÓW***************
bStateError:= (eState=E_Station.eError) OR (eState=E_Station.eResetting) OR bIgnoreError;




IF bEnable THEN
	
	//Error 1 - Blokada otwarcia chwytaka
	tonOpeningBlocked(IN:=NOT bCatchActuator AND NOT bOpenedActuatorSensor, PT:=T#3S);
	
	IF tonOpeningBlocked.Q AND NOT bStateError THEN
		sErrorDescription:='Blokada otwarcia chwytaka - sprawdź czujnik';
		bHeightMotorUp:=FALSE;
		bError := TRUE;
		nErrorNr:=281;	
		//nErrorNr := nErrorNr+iStationIndex;
	END_IF
	
	//Error 2 - podnośnik nie porusza się pomimo wysterowania 
	tonErrorHeightChange(IN:=(bHeightMotorUp OR bHeightMotorDown) AND nLastPositionHeightCV=lrHeightMotorCV AND NOT bNoLifter, PT:=T#3S);
	
	IF tonErrorHeightChange.Q AND NOT bStateError THEN
		bHeightMotorUp:=FALSE;
		bHeightMotorDown:=FALSE;
		bError := TRUE;
		nErrorNr:=282;
		//nErrorNr := nErrorNr+iStationIndex;
		sErrorDescription:='Blokada podnośnika lub brak zasilania - sprawdź czujnik lub odblokuj mechanicznie';	
	END_IF
	
	
	//Error 3 - Bład nastaw max
	tonMaxHeight(IN:=nPositionHeightSV>lrMaxHeight+1 AND bHomingDone AND lrMaxHeight>0 AND eState=E_Station.eReady,PT:=T#30S);
	IF tonMaxHeight.Q AND NOT bStateError THEN
		bHeightMotorUp:=FALSE;
		bHeightMotorDown:=FALSE;
		bError := TRUE;
		nErrorNr:=283;
		//nErrorNr := nErrorNr+iStationIndex;
		sErrorDescription:='Wartość zadana wysokości jest większa od maksymalnej - zmień ustawienia w recepturze';
		sErrorDescription2:=REAL_TO_STRING(LREAL_TO_INT(lrMaxHeight));
	END_IF
	
	//Error 4 - Bład nastaw min
	tonMinHeight(IN:=nPositionHeightSV<lrMinHeight-1 AND bHomingDone AND lrMinHeight>0 AND eState=E_Station.eReady,PT:=T#30S);
	IF tonMinHeight.Q AND NOT bStateError THEN
		bHeightMotorUp:=FALSE;
		bHeightMotorDown:=FALSE;
		bError := TRUE;
		nErrorNr:=284;
		//nErrorNr := nErrorNr+iStationIndex;
		sErrorDescription:='Wartość zadana wysokości jest mniejsza od minimalnej - zmień ustawienia w recepturze ';
		sErrorDescription2:=REAL_TO_STRING(LREAL_TO_INT(lrMinHeight));
	END_IF
	
	//Error 5 - Bład zbyt dużej różnicy nastaw
	//tonSVCVDiffHeight(IN:=ABS(nPositionHeightSV-lrHeightMotorCV)>10 AND bHomingDone AND NOT bAlarmSVCVDiffHeightDisable AND eState=E_Station.eReady AND NOT bChangeOver2,PT:=T#5M);
	IF tonSVCVDiffHeight.Q AND NOT bStateError THEN
		bHeightMotorUp:=FALSE;
		bHeightMotorDown:=FALSE;
		bError := TRUE;
		nErrorNr:=285;
		//nErrorNr := nErrorNr+iStationIndex;
		sErrorDescription:='Wartość aktualna jest zbyt różna od zadanej - zmień ustawienia w recepturze lub ustaw stację';
		sErrorDescription2:=REAL_TO_STRING(LREAL_TO_INT(nPositionHeightSV));
		
	END_IF	
		
	
	
ELSE
	bError := FALSE;
END_IF

	
//******************PRZEJŚCIE DO eERROR*****************************

IF bError AND NOT bStateError THEN
	IF eLastState = eRunning THEN
		bCycleNotDone := TRUE;
	END_IF
	eState := E_Station.eError;
END_IF

//****************WYŚWIETLANIE STATUSU BLEDU***********************

(*Wyświetlanie błedu na wyjściu*)
bError;

(*Przepisywanie nazwy stacji*)
sErrorStationName := sStationName;


//Jezeli nie zbazowane to potrzebne bazowanie
IF NOT bHeightMotorEncoderHomed AND NOT bNoLifter  THEN
	bHomingDone:=FALSE;
END_IF
END_ACTION

ACTION HeightMotor:
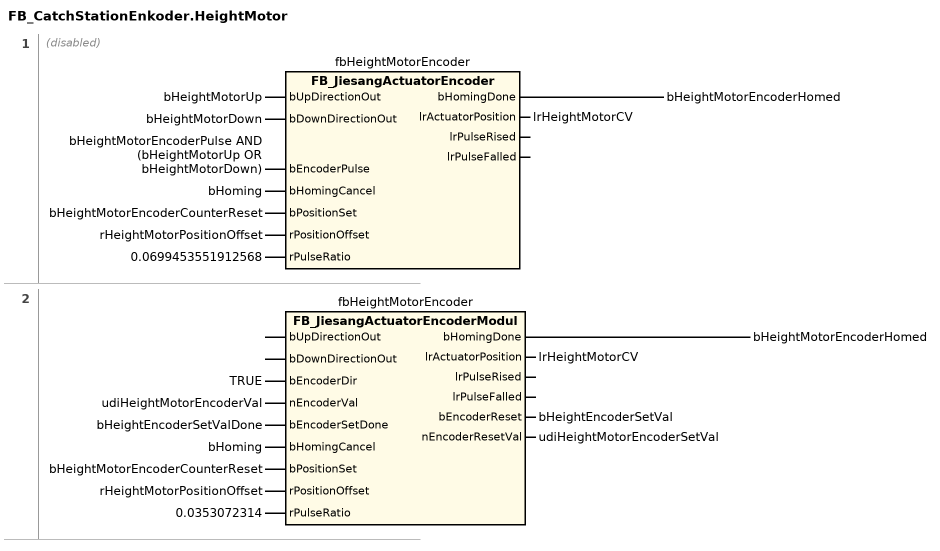
// NETWORK 1 (disabled)
// fbHeightMotorEncoder(
//     bUpDirectionOut := bHeightMotorUp,
//     bDownDirectionOut := bHeightMotorDown,
//     bEncoderPulse := bHeightMotorEncoderPulse AND (bHeightMotorUp OR bHeightMotorDown),
//     bHomingCancel := bHoming,
//     bPositionSet := bHeightMotorEncoderCounterReset,
//     rPositionOffset := rHeightMotorPositionOffset,
//     rPulseRatio := 0.0699453551912568,
//     lrActuatorPosition => lrHeightMotorCV); // FB_JiesangActuatorEncoder
// bHeightMotorEncoderHomed := fbHeightMotorEncoder.bHomingDone;

// NETWORK 2
fbHeightMotorEncoder(
    bEncoderDir := TRUE,
    nEncoderVal := udiHeightMotorEncoderVal,
    bEncoderSetDone := bHeightEncoderSetValDone,
    bHomingCancel := bHoming,
    bPositionSet := bHeightMotorEncoderCounterReset,
    rPositionOffset := rHeightMotorPositionOffset,
    rPulseRatio := 0.0353072314,
    lrActuatorPosition => lrHeightMotorCV,
    bEncoderReset => bHeightEncoderSetVal,
    nEncoderResetVal => udiHeightMotorEncoderSetVal); // FB_JiesangActuatorEncoderModul
bHeightMotorEncoderHomed := fbHeightMotorEncoder.bHomingDone;
END_ACTION

ACTION Homing:
//BAZOWANIE
bCatchActuator:=FALSE;
	
//Uwaga nie zmieniać czasu bo jednocześnie dwie stację jadą do góry
tofHeightMotorDown(IN:=bHeightMotorDown, PT:=T#1S); //Zabezpieczenie przed zbyt szybkim przełączeniem pomiędzy Down a Up, bezpiecznieki sie palą, 


//Podnoszenie stacji do maksymalnej pozycji
IF NOT bHeightMotorEncoderHomed OR rtEncoderHomed.Q THEN
	bHeightMotorUp:=(*TRUE*) NOT tofHeightMotorDown.Q;;
	bHeightMotorDown:=FALSE;
	IF tonHeightNoChange.Q THEN
		bHeightMotorEncoderCounterReset:=TRUE;
		bHeightMotorUp:=FALSE;
	END_IF
	//Jesli enkoder zbazowany zakończ bazowanie	
	IF rtEncoderHomed.Q THEN
		bHeightMotorUp:=FALSE;
		bHeightMotorDown:=FALSE;
		eState:=E_Station.eHomingDone;
	END_IF		
		
//Po podniesieniu stacji opuszczanie do ustalonej wysokości
ELSIF bHeightMotorEncoderHomed THEN
	bHeightMotorEncoderCounterReset:=FALSE;
	bHeightMotorUp:=lrHeightMotorCV<=nPositionHeightSV;
	bHeightMotorDown:=lrHeightMotorCV>=nPositionHeightSV (*AND lrHeightMotorCV>=lrMinHeight*);
	//Kiedy stacja osiągnie wysokość zadaną
	IF ABS(lrHeightMotorCV-nPositionHeightSV)<0.6 OR tonLimitPosMaxReachedDelay.Q OR tonLimitPosMinReachedDelay.Q (*OR lrHeightMotorCV>=lrMinHeight*) THEN
		bHeightMotorDown:=FALSE;
		bHeightMotorUp:=FALSE;
		eState:=E_Station.eHomingDone;
	END_IF			
END_IF

	
//Opcja braku podnośnika	
IF bNoLifter THEN
	eState:=E_Station.eHomingDone;
END_IF
END_ACTION

ACTION ManualMovements:

//W trybie ruchów manualnych wykonuj ruchy za pomocą rozkazów manualnych
IF NOT bRun THEN
	bCatchActuator:=bManualCatchActuator;
	bHeightMotorUp:=bManualHeightMotorUp;
	bHeightMotorDown:=bManualHeightMotorDown;
ELSE	//Kasuje zeby po cyklu nic sie nie poruszało
	bManualCatchActuator := FALSE;
	bManualHeightMotorUp  := FALSE;
	bManualHeightMotorDown  := FALSE;
END_IF


IF bHoming OR bHeightSet THEN
	eState:=E_Station.eHoming;
END_IF
	
Running();
	
//Zabezpieczenie przed kolizją stacji poprzez ruch podnośnika	
IF bHeightMotorDown AND lrHeightMotorCV<=lrMinHeight AND NOT bHoming AND NOT bHeightSet THEN
	bHeightMotorDown:=FALSE;
END_IF	

IF bHeightMotorUp AND lrHeightMotorCV>=lrMaxHeight AND NOT bHoming AND NOT bHeightSet THEN
	bHeightMotorUp:=FALSE;
END_IF		 

IF NOT bRun THEN
	bCycleDone 					:= FALSE;
	bCycleNotDone 				:= FALSE;	
END_IF
END_ACTION

ACTION Running:

//Timery
tonCatchingTime(IN:=(eRunningState=E_CatchStationState.eCatching), PT:=T#500MS);


CASE eRunningState OF
	
	//NIEGOTOWY
	E_CatchStationState.eDisabled:
		eRunningState:=E_CatchStationState.eReady;

	//Chwytak gotowy do pracy
	E_CatchStationState.eReady: 
		//Jeśli komenda chwytania przejdz do stanu chwytanie
		IF NOT bCycleDone AND NOT bCycleNotDone THEN
			IF bRun THEN
			eRunningState:=E_CatchStationState.eCatching;
			END_IF
		END_IF
		
	//Chwytanie 
	E_CatchStationState.eCatching:
		bCatchActuator:=TRUE;
		

		IF tonCatchingTime.Q THEN
			IF bClosedActuatorSensor THEN
				eRunningState	:= E_CatchStationState.eCatched;
			ELSE
				eRunningState	:= E_CatchStationState.eNotCatched;
			END_IF
		END_IF

	//Uchwycone 
	E_CatchStationState.eCatched:
		bCatchActuator:=bRun;
		bCycleDone := TRUE;
		//Kiedy zniknie rozkaz chwytania i 
	
	E_CatchStationState.eNotCatched:
	
		bCatchActuator:=bRun;                                   
		bCycleDone := TRUE;
	
END_CASE
END_ACTION

ACTION Statistics:



rtrigCycleTimerRead(CLK:=eRunningState=E_CatchStationState.eCatched);
IF rtrigCycleTimerRead.Q THEN
	tCycleTime:=tonCycleTimer.ET;
END_IF
tonCycleTimer(IN:=eState>E_Station.eReady,PT:=T#1D);
END_ACTION

END_FUNCTION_BLOCK

// ---- POUs/FB/FB_CatchStationEnkoder_old.TcPOU
(*
Nazwa:			FB_CatchStation
Opis:			Chwytak pod stacjami 
Wersja:			v1.1
Data:			2023-02-22
Autor:			TW,DP
Urzadzenia:		Silownik chwytania, podnośnik JIESANG
Konfiguracja:	
Zmiany:
20230222 - Zwieksozmny czas bledu 9
Info:
- dodano błędy od nastaw powyżej max i min (error 7 i 8)
- dodawno bHomingNeeded
- wylaczanie wyjść zmiana 2 wylaczanie wyjsc jak zniknie Enable
*)


FUNCTION_BLOCK FB_CatchStationEnkoder_old
VAR_INPUT
	bEnable: BOOL;						//Zezwolenie na pracę
	bEStop:BOOL;						//Stop Awaryjny włączony
	bRun:BOOL;							//Rozkaz łapania 
	bHoming:BOOL;						//Zezwolenie na wykonanie bazowania i pozycjonowania podajnika
	bHeightSet:BOOL;					//Ustaw wysokość
	bChangeover:BOOL;					//Ustawianie na zadaną wysokość do wymiany elementów formatowych
	bChangeOver2:BOOL;
	bIgnoreError:BOOL;					//Ignorowania błędów cyklu pracy
	bReset:BOOL;						//Reset błędu, jeśli w stanie "eError"
	nGripperScrewerPosition   	:LREAL; // Aktualna pozycja serwa od podnoszenia
	nSafetyScrewerPosition		:LREAL;	// zadana bezpieczna pozycja 
	bScrewerbError				:BOOL;  // Sygnał błędu od zakręcarki
	nPositionHeightSV:LREAL;			//Wysokość zadana na której ma znajdować się stacja
	bOpenedActuatorSensor:BOOL;			//Czujnik otwarcia siłownika łapania
	bClosedActuatorSensor:BOOL;			//Czujnik otwarcia siłownika łapania
	lrMaxHeight:LREAL;					//Maksymalna wysokość podnośnika chwytaka
	lrMinHeight:LREAL;					//Minimalna wysokość podnośnika chwytaka
	bManualMovement:BOOL;				//Zezwolenie na ruchy ręcznę
	bUnlockColision:BOOL:=FALSE;		//Odblokowywanie możliwośći kolizji
	bAlarmSVCVDiffHeightDisable:BOOL;	//Wyłączenie alarmu od rożnicy wysokości zadanej od aktualnej
	bNoLifter:BOOL;						//Podnośnik
	
	_HEIGHTMOTOR_ 				:BOOL;
	udiHeightMotorEncoderVal	:UDINT;		//Ilość impulsów z modułu enkoderowego
	bHeightEncoderSetValDone	:BOOL;		//Zerowanie enkodera wykonane
	bHeightMotorEncoderPulse 	:BOOL;			//Sygnał impulsów enkodera siłownika
	rHeightMotorPositionOffset 	:REAL;		//Wysokość bazowani podnośnika

	_ALARMINFO_ :BOOL;
	iStationIndex:UDINT;					//Numer stacji 
	sStationName:STRING;					//Nazwa stacji	

	
END_VAR
VAR_OUTPUT
	eState: E_Station;						//Stan ogólny bloku
	eRunningState: E_CatchStationState;		//Stan wewnętrzny
	bError: BOOL;							//Błąd stacji
	nErrorNr: UDINT;						//Nr błędu podajnika platynek
	sErrorDescription:STRING(200);				//Opis błędu
	sErrorDescription2: STRING(200);				//Opis błędu 2
	sErrorStationName:STRING;				//Nazwa stacji
	udiStationID: UDINT;				// Nr stacji

	bCatchActuator:BOOL;					//Sterownie siłownika łapania opakowania
	bHeightMotorUp:BOOL;					//Sterowanie silnikiem podnośnika  - RUCH W GÓRĘ
	bHeightMotorDown:BOOL;					//Sterowanie silnikiem podnośnika  - RUCH W DÓŁ
	udiHeightMotorEncoderSetVal	:UDINT;		
	bHeightEncoderSetVal	:BOOL;		//Zerowanie enkodera
	lrHeightMotorCV:LREAL;					//Aktualna pozycja podnośnika
	tCycleTime:TIME;
	bHomingDone:BOOL;						//Wymagane ponowne bazowanie (blad podczas bazowania lub stop awaryjny)
	bCycleDone:BOOL;
	bCycleNotDone:BOOL;
END_VAR
VAR
	tonHeightNoChange: TON; 			//Timer wykrycia braku ruchu siłownika zmiany wysokości stacji
	nLastPositionHeightCV: LREAL;		//Pozycja podnośnika w poprzednim cyklu programu
	tonErrorHeightChange: TON; 			//Timer błędu podnośnika
	// Czas zadziałania siłownika
	tonCatchingTime: TON;
	// Timer blokady otwierania chwytaka
	tonOpeningBlocked: TON;
	rtEncoderHomed:R_TRIG;
	tonCycleTimer:TON;
	rtrigCycleTimerRead:R_TRIG;
	
	tofMotorUpPermition: TOF;
	tofMotorDownPermition: TOF;
	tonLimitPosMinReachedDelay: TON;
	tonLimitPosMaxReachedDelay: TON;
	tonMaxHeight		: TON;
	tonMinHeight		: TON;
	tonSVCVDiffHeight	: TON;
	
	//Podnośnik Jiesang	
	fbHeightMotorEncoder: FB_JiesangActuatorEncoderModul;//FB_JiesangActuatorEncoder;	// Blok enkodera podnośnika chwytaka stabilizującego pod zakręcarką	
	bHeightMotorEncoderCounterReset:BOOL; 				//Sygnał resetu enkodera
	bHeightMotorEncoderHomed:BOOL;						//Informacja od enkodera że jest zbazowany

	eLastState: E_Station;							//Stan ogólny bloku
	eLastRunningState: E_CatchStationState;			//Stan podbloku
	eLastStateTemp: E_Station;						//Stan ogólny bloku
	eLastRunningStateTemp: E_CatchStationState;		//Stan podbloku
	bStateError: BOOL;

	tonStopping: TON;
	tofHeightMotorDown: TOF;
	iCaseChangeover: INT;
	tonChangeOverLimitPosMinReachedDelay: TON;
	tonChangeoverLimitPosMaxReachedDelay: TON;
END_VAR

VAR_IN_OUT
	bManualCatchActuator:BOOL;		//Ruch ręczny siłownikiem podajnika platynek
	bManualHeightMotorUp:BOOL;			//Ruch ręczny podnośnika stacji w górę
	bManualHeightMotorDown:BOOL;		//Ruch ręczny podnośnika stacji w dół
END_VAR

HeightMotor();
ErrorHandling();
Control();
Changeover();
Statistics();
aStationID();
(*Zapisywanie ostatniego stanu*)
IF eLastStateTemp<>eState THEN
	eLastState := eLastStateTemp;
END_IF
eLastStateTemp := eState;
IF eLastRunningStateTemp<>eRunningState THEN
	eLastRunningState := eLastRunningStateTemp;
END_IF
eLastRunningStateTemp := eRunningState;
(*Koniec Zapisywanie ostatniego stanu*)


nLastPositionHeightCV:=lrHeightMotorCV;

ACTION aStationID:
udiStationID	:=	iStationIndex;
END_ACTION

ACTION Changeover:
tonChangeOverLimitPosMinReachedDelay(IN:=(lrHeightMotorCV<=lrMinHeight) AND bChangeover,PT:=T#2S);
tonChangeoverLimitPosMaxReachedDelay(IN:=(lrHeightMotorCV>=lrMaxHeight) AND bChangeover,PT:=T#2S);


//Przeniesione do PreparingToDisabled
(*CASE iCaseChangeover OF
	
	0: //Włączenie ustawiania
		IF bChangeover THEN
			iCaseChangeover := iCaseChangeover + 10;
			bHeightMotorDown:=FALSE;
			bHeightMotorUp:=FALSE;
		END_IF
		
	10: //Ustawianie stacji na wysokość 
		IF bHeightMotorEncoderHomed THEN
			bHeightMotorEncoderCounterReset	:=	FALSE;
			bHeightMotorUp					:=	lrHeightMotorCV	<=	200;
			bHeightMotorDown				:=	lrHeightMotorCV	>=	200;
			//Kiedy stacja osiągnie wysokość zadaną
			IF ABS(lrHeightMotorCV-nPositionHeightSV)<2 OR tonChangeoverLimitPosMaxReachedDelay.Q OR tonChangeOverLimitPosMinReachedDelay.Q  THEN
				bHeightMotorDown			:=	FALSE;
				bHeightMotorUp				:=	FALSE;
				iCaseChangeover 			:=	iCaseChangeover + 10;
			END_IF			
		ELSE
			bHeightMotorDown		:=	FALSE;
			bHeightMotorUp			:=	FALSE;
			iCaseChangeover 		:=  0;
		END_IF	
		
	20: //Czekanie na wyłączenie przezbrajania i ustawienie na odpowiednią wysokość z receptury
			IF NOT bChangeover THEN
				iCaseChangeover := iCaseChangeover + 10;
			END_IF
	30: //Ustawianie stacji na wysokość z receptury
		IF bHeightMotorEncoderHomed THEN
			bHeightMotorEncoderCounterReset	:=	FALSE;
			bHeightMotorUp					:=	lrHeightMotorCV	<=	nPositionHeightSV;
			bHeightMotorDown				:=	lrHeightMotorCV	>=	nPositionHeightSV;
			//Kiedy stacja osiągnie wysokość zadaną
			IF ABS(lrHeightMotorCV-nPositionHeightSV)<2 OR tonChangeoverLimitPosMaxReachedDelay.Q OR tonChangeOverLimitPosMinReachedDelay.Q  THEN
				bHeightMotorDown			:=	FALSE;
				bHeightMotorUp				:=	FALSE;
				iCaseChangeover 			:=	iCaseChangeover + 10;
			END_IF			
		ELSE
			bHeightMotorDown		:=	FALSE;
			bHeightMotorUp			:=	FALSE;
			iCaseChangeover 		:=  0;
		END_IF
	40: //Ustawianie stacji na wysokość z receptury	
		iCaseChangeover 		:=  0;

END_CASE
*)
END_ACTION

ACTION Control:

	(** TIMERY**)
	rtEncoderHomed(CLK:=bHeightMotorEncoderHomed,Q=>);
	tonHeightNoChange(IN:=((bHeightMotorUp OR bHeightMotorDown) AND (nLastPositionHeightCV=lrHeightMotorCV)), PT:=T#1S); 
	tonLimitPosMinReachedDelay(IN:=(lrHeightMotorCV<=lrMinHeight) AND eState=E_Station.eHoming,PT:=T#2S);
	tonLimitPosMaxReachedDelay(IN:=(lrHeightMotorCV>=lrMaxHeight) AND eState=E_Station.eHoming,PT:=T#2S);
	tonStopping(IN:=eState=E_Station.eStopping,PT:=T#2S);
	tofMotorUpPermition(IN:=bHeightMotorDown,PT:=T#250MS);
	tofMotorDownPermition(IN:=bHeightMotorUp ,PT:=T#250MS);	
	(*****Wyłączenie enable*****)
	IF NOT bEnable OR bChangeover THEN //Lub przezbrajania
		IF eState <> E_Station.eDisabled AND eState <> E_Station.ePreparingToDisable AND nGripperScrewerPosition>nSafetyScrewerPosition AND NOT bScrewerbError THEN
				eState 				:= E_Station.ePreparingToDisable; 
		END_IF	
	END_IF

	(*****Estop*****)
	IF NOT bEstop  THEN	
		IF eState <> E_Station.eAborted AND eState <> E_Station.eAborting AND eState <> E_Station.eDisabled THEN
				eState 				:= E_Station.eAborting; 
		END_IF
	END_IF

	CASE eState OF
	/////////////////////////////	
		E_Station.eDisabled: 					// Stan nieaktywnosci (Stacja wyłączona) 

			IF bEnable THEN
				eState 				:= E_Station.ePreparingToReady; 
			END_IF 
			
    /////////////////////////////	    
		E_Station.eAborted: 					// Stan bezpiecznego zatrzymania (po Abortingu) 

			IF bEStop THEN
				eState 				:= E_Station.ePreparingToReady;
			END_IF
			
	/////////////////////////////	
		E_Station.eAborting:                 	// Stan bezpiecznego zatrzymywania (po EStopie)

			bHeightMotorUp				:=	FALSE;
			bHeightMotorDown			:=	FALSE;
			eState := E_Station.eAborted;  
			eRunningState:=E_CatchStationState.eDisabled;
			
	/////////////////////////////			
		E_Station.eError:                 	 	// Stan błędu 	

			iCaseChangeover 		:=	0;
			IF bReset THEN
				eState 				:=	E_Station.eResetting;
			END_IF
						
	/////////////////////////////
		E_Station.eResetting:					// Stan resetowania bledu (po Errorze)
	
			bError := FALSE;

			IF NOT bError THEN
				nErrorNr 			:=	0;
   				sErrorDescription 	:=	'';
				eState 				:=	E_Station.ePreparingToReady;
			ELSE
				eState 				:=	E_Station.eError;
			END_IF
        
	/////////////////////////////
		E_Station.eManualMovement:     			// Stan ruchów manualnych  

			ManualMovements();
			//Wyjście z trybu serwisowego
			IF NOT bManualMovement THEN
				bCatchActuator				:=	FALSE;
				bHeightMotorUp				:=	FALSE;
				bHeightMotorDown			:=	FALSE;
				bManualCatchActuator		:=	bCatchActuator;
				eState:=E_Station.eReady;
			END_IF

	/////////////////////////////
		E_Station.eHoming:						// Stan bazowania 
	IF (nGripperScrewerPosition>nSafetyScrewerPosition AND NOT bScrewerbError) OR bManualMovement THEN  // co to za bzdura
			Homing();
			IF NOT bHoming AND NOT bHeightSet THEN // co to za bzdura
			   eState:=E_Station.ePreparingToReady;
			   	bHeightMotorDown:=FALSE;
				bHeightMotorUp:=FALSE;
			END_IF		
	END_IF		
	/////////////////////////////
		E_Station.eHomingDone:                  // Stan wykonania bazowania 
	
			bHeightMotorDown					:=	FALSE;
			bHeightMotorUp						:=	FALSE;
			bHeightMotorEncoderCounterReset		:=	FALSE;
			bHomingDone							:=	TRUE;
			IF NOT bHoming AND NOT bHeightSet THEN
			   eState:=E_Station.eReady;
			END_IF
			
	/////////////////////////////
		E_Station.ePreparingToReady:            // Stan przygotowywania do gotowosci (zawsze przed Ready)  
	
			bCatchActuator	:=	FALSE;
			eRunningState	:=	E_CatchStationState.eReady;
			eState			:=	E_Station.eReady;	
			
	/////////////////////////////
		E_Station.ePreparingToDisable:          // Stan przygotowywania do nieaktywnosci (po wyłączeniu Enable) 
  
			bCatchActuator:=FALSE;
			IF NOT bChangeOver THEN //Normalne wyłączenie
				bHeightMotorUp:=TRUE;
				bHeightMotorDown:=FALSE;	
				IF tonHeightNoChange.Q THEN
					bHeightMotorUp:=FALSE;
					eState:=E_Station.eDisabled;
					eRunningState:=E_CatchStationState.eDisabled;
				END_IF	
			ELSE //Wyłączenie z przebrajaniem na pozycje 200
				IF bHeightMotorEncoderHomed THEN
					bHeightMotorEncoderCounterReset	:=	FALSE;
					bHeightMotorUp					:=	lrHeightMotorCV	<=	150 AND NOT tofMotorUpPermition.Q;
					bHeightMotorDown				:=	lrHeightMotorCV	>=	150 AND NOT tofMotorDownPermition.Q;
					//Kiedy stacja osiągnie wysokość zadaną
					IF ABS(lrHeightMotorCV-150)<2 OR tonChangeoverLimitPosMaxReachedDelay.Q OR tonChangeOverLimitPosMinReachedDelay.Q  THEN
						bHeightMotorDown			:=	FALSE;
						bHeightMotorUp				:=	FALSE;
						eState						:=	E_Station.eDisabled;
						eRunningState				:=	E_CatchStationState.eDisabled;
					END_IF			
				ELSE
					bHeightMotorDown				:=	FALSE;
					bHeightMotorUp					:=	FALSE;
					eState								:=E_Station.eDisabled;
					eRunningState					:=	E_CatchStationState.eDisabled;
				END_IF	
			END_IF
				
	/////////////////////////////
		E_Station.eReady:						// Stan gotowosci 

			IF bRun AND NOT bCycleDone AND NOT bCycleNotDone THEN
				eState 				:= E_Station.eStarting; 
			END_IF
			IF bHoming OR bHeightSet OR bChangeover THEN
				eState 				:= E_Station.eHoming; 
			END_IF
			IF bManualMovement THEN
				//Jeśli przejście w tryb ruchów manualnych przepisz wszystkie stany siłowników sterowanych przez moduł
				//aby zapobiec ewentualnym kolizjom po wejściu w tryb serwisowy
				bManualCatchActuator		:= bCatchActuator;
				bManualHeightMotorUp		:= bHeightMotorUp;
				bManualHeightMotorDown		:= bHeightMotorDown;
				
				eState 						:= E_Station.eManualMovement; 
				eRunningState 				:= E_CatchStationState.eReady;
 
			END_IF
			IF NOT bRun THEN
				bCycleDone 			:= FALSE;
				bCycleNotDone 		:= FALSE;			
			END_IF
			
	/////////////////////////////
		E_Station.eStopping:					// Stan zatrzymywania 
					
			Running();
			IF bOpenedActuatorSensor OR tonStopping.Q THEN //NEW
				eState						:=	E_Station.eReady;
				eRunningState 				:=	E_CatchStationState.eReady;
			END_IF
			
	/////////////////////////////
		E_Station.eStarting:                  	// Stan uruchamiania (po Ready)
				
			eState					 := E_Station.eRunning; 

	/////////////////////////////
		E_Station.eRunning:               		// Stan wykonywania cyklu (po Startingu), w tym stanie osobny

			Running();
			IF NOT bRun THEN 					(*Przerywanie cyklu*)
				eState				:= E_Station.eStopping;
				bCycleNotDone		:= TRUE;
			END_IF
			(*IF bCycleDone OR bCycleNotDone THEN (*Cykl zakończony*)
				eState 				 := E_Station.eReady;
			END_IF*)						
		ELSE
		
		
	/////////////////////////////		
	END_CASE
END_ACTION

ACTION ErrorHandling:
//OBSŁUGA BŁĘDÓW PODAJNIKA PLATYNEK

//************LISTA BŁĘDÓW***************
bStateError:= (eState=E_Station.eError) OR (eState=E_Station.eResetting) OR bIgnoreError;




IF bEnable THEN
	
	//Error 1 - Blokada otwarcia chwytaka
	tonOpeningBlocked(IN:=NOT bCatchActuator AND NOT bOpenedActuatorSensor, PT:=T#3S);
	
	IF tonOpeningBlocked.Q AND NOT bStateError THEN
		sErrorDescription:='Blokada otwarcia chwytaka - sprawdź czujnik';
		bHeightMotorUp:=FALSE;
		bError := TRUE;
		nErrorNr:=281;	
		//nErrorNr := nErrorNr+iStationIndex;
	END_IF
	
	//Error 2 - podnośnik nie porusza się pomimo wysterowania 
	tonErrorHeightChange(IN:=(bHeightMotorUp OR bHeightMotorDown) AND nLastPositionHeightCV=lrHeightMotorCV AND NOT bNoLifter, PT:=T#3S);
	
	IF tonErrorHeightChange.Q AND NOT bStateError THEN
		bHeightMotorUp:=FALSE;
		bHeightMotorDown:=FALSE;
		bError := TRUE;
		nErrorNr:=282;
		//nErrorNr := nErrorNr+iStationIndex;
		sErrorDescription:='Blokada podnośnika lub brak zasilania - sprawdź czujnik lub odblokuj mechanicznie';	
	END_IF
	
	
	//Error 3 - Bład nastaw max
	tonMaxHeight(IN:=nPositionHeightSV>lrMaxHeight+1 AND bHomingDone AND lrMaxHeight>0 AND eState=E_Station.eReady,PT:=T#30S);
	IF tonMaxHeight.Q AND NOT bStateError THEN
		bHeightMotorUp:=FALSE;
		bHeightMotorDown:=FALSE;
		bError := TRUE;
		nErrorNr:=283;
		//nErrorNr := nErrorNr+iStationIndex;
		sErrorDescription:='Wartość zadana wysokości jest większa od maksymalnej - zmień ustawienia w recepturze';
		sErrorDescription2:=REAL_TO_STRING(LREAL_TO_INT(lrMaxHeight));
	END_IF
	
	//Error 4 - Bład nastaw min
	tonMinHeight(IN:=nPositionHeightSV<lrMinHeight-1 AND bHomingDone AND lrMinHeight>0 AND eState=E_Station.eReady,PT:=T#30S);
	IF tonMinHeight.Q AND NOT bStateError THEN
		bHeightMotorUp:=FALSE;
		bHeightMotorDown:=FALSE;
		bError := TRUE;
		nErrorNr:=284;
		//nErrorNr := nErrorNr+iStationIndex;
		sErrorDescription:='Wartość zadana wysokości jest mniejsza od minimalnej - zmień ustawienia w recepturze ';
		sErrorDescription2:=REAL_TO_STRING(LREAL_TO_INT(lrMinHeight));
	END_IF
	
	//Error 5 - Bład zbyt dużej różnicy nastaw
	//tonSVCVDiffHeight(IN:=ABS(nPositionHeightSV-lrHeightMotorCV)>10 AND bHomingDone AND NOT bAlarmSVCVDiffHeightDisable AND eState=E_Station.eReady AND NOT bChangeOver2,PT:=T#5M);
	IF tonSVCVDiffHeight.Q AND NOT bStateError THEN
		bHeightMotorUp:=FALSE;
		bHeightMotorDown:=FALSE;
		bError := TRUE;
		nErrorNr:=285;
		//nErrorNr := nErrorNr+iStationIndex;
		sErrorDescription:='Wartość aktualna jest zbyt różna od zadanej - zmień ustawienia w recepturze lub ustaw stację';
		sErrorDescription2:=REAL_TO_STRING(LREAL_TO_INT(nPositionHeightSV));
		
	END_IF	
		
	
	
ELSE
	bError := FALSE;
END_IF

	
//******************PRZEJŚCIE DO eERROR*****************************

IF bError AND NOT bStateError THEN
	IF eLastState = eRunning THEN
		bCycleNotDone := TRUE;
	END_IF
	eState := E_Station.eError;
END_IF

//****************WYŚWIETLANIE STATUSU BLEDU***********************

(*Wyświetlanie błedu na wyjściu*)
bError;

(*Przepisywanie nazwy stacji*)
sErrorStationName := sStationName;


//Jezeli nie zbazowane to potrzebne bazowanie
IF NOT bHeightMotorEncoderHomed AND NOT bNoLifter  THEN
	bHomingDone:=FALSE;
END_IF
END_ACTION

ACTION HeightMotor:
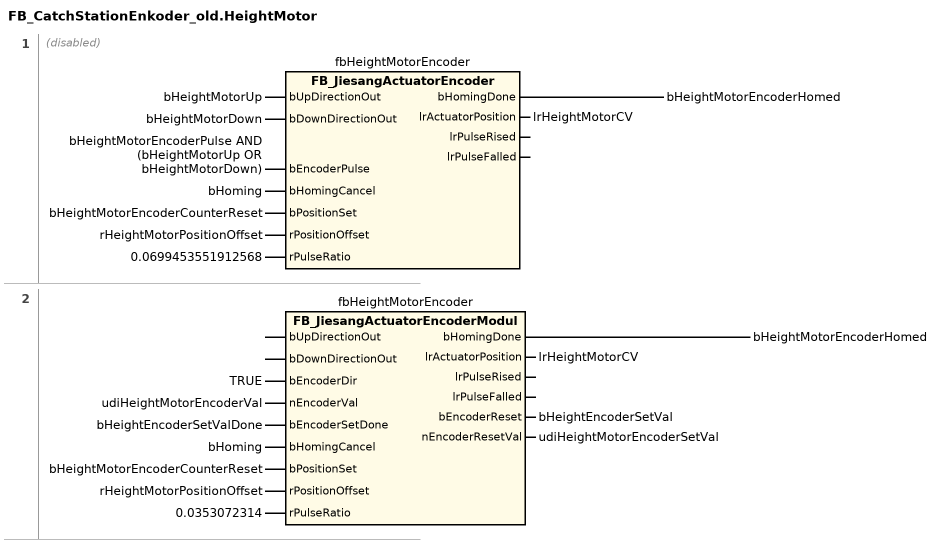
// NETWORK 1 (disabled)
// fbHeightMotorEncoder(
//     bUpDirectionOut := bHeightMotorUp,
//     bDownDirectionOut := bHeightMotorDown,
//     bEncoderPulse := bHeightMotorEncoderPulse AND (bHeightMotorUp OR bHeightMotorDown),
//     bHomingCancel := bHoming,
//     bPositionSet := bHeightMotorEncoderCounterReset,
//     rPositionOffset := rHeightMotorPositionOffset,
//     rPulseRatio := 0.0699453551912568,
//     lrActuatorPosition => lrHeightMotorCV); // FB_JiesangActuatorEncoder
// bHeightMotorEncoderHomed := fbHeightMotorEncoder.bHomingDone;

// NETWORK 2
fbHeightMotorEncoder(
    bEncoderDir := TRUE,
    nEncoderVal := udiHeightMotorEncoderVal,
    bEncoderSetDone := bHeightEncoderSetValDone,
    bHomingCancel := bHoming,
    bPositionSet := bHeightMotorEncoderCounterReset,
    rPositionOffset := rHeightMotorPositionOffset,
    rPulseRatio := 0.0353072314,
    lrActuatorPosition => lrHeightMotorCV,
    bEncoderReset => bHeightEncoderSetVal,
    nEncoderResetVal => udiHeightMotorEncoderSetVal); // FB_JiesangActuatorEncoderModul
bHeightMotorEncoderHomed := fbHeightMotorEncoder.bHomingDone;
END_ACTION

ACTION Homing:
//BAZOWANIE
bCatchActuator:=FALSE;
	
//Uwaga nie zmieniać czasu bo jednocześnie dwie stację jadą do góry
tofHeightMotorDown(IN:=bHeightMotorDown, PT:=T#1S); //Zabezpieczenie przed zbyt szybkim przełączeniem pomiędzy Down a Up, bezpiecznieki sie palą, 


//Podnoszenie stacji do maksymalnej pozycji
IF NOT bHeightMotorEncoderHomed OR rtEncoderHomed.Q THEN
	bHeightMotorUp:=(*TRUE*) NOT tofHeightMotorDown.Q;;
	bHeightMotorDown:=FALSE;
	IF tonHeightNoChange.Q THEN
		bHeightMotorEncoderCounterReset:=TRUE;
		bHeightMotorUp:=FALSE;
	END_IF
	//Jesli enkoder zbazowany zakończ bazowanie	
	IF rtEncoderHomed.Q THEN
		bHeightMotorUp:=FALSE;
		bHeightMotorDown:=FALSE;
		eState:=E_Station.eHomingDone;
	END_IF		
		
//Po podniesieniu stacji opuszczanie do ustalonej wysokości
ELSIF bHeightMotorEncoderHomed THEN
	bHeightMotorEncoderCounterReset:=FALSE;
	bHeightMotorUp:=lrHeightMotorCV<=nPositionHeightSV;
	bHeightMotorDown:=lrHeightMotorCV>=nPositionHeightSV (*AND lrHeightMotorCV>=lrMinHeight*);
	//Kiedy stacja osiągnie wysokość zadaną
	IF ABS(lrHeightMotorCV-nPositionHeightSV)<0.6 OR tonLimitPosMaxReachedDelay.Q OR tonLimitPosMinReachedDelay.Q (*OR lrHeightMotorCV>=lrMinHeight*) THEN
		bHeightMotorDown:=FALSE;
		bHeightMotorUp:=FALSE;
		eState:=E_Station.eHomingDone;
	END_IF			
END_IF

	
//Opcja braku podnośnika	
IF bNoLifter THEN
	eState:=E_Station.eHomingDone;
END_IF
END_ACTION

ACTION ManualMovements:

//W trybie ruchów manualnych wykonuj ruchy za pomocą rozkazów manualnych
IF NOT bRun THEN
	bCatchActuator:=bManualCatchActuator;
	bHeightMotorUp:=bManualHeightMotorUp;
	bHeightMotorDown:=bManualHeightMotorDown;
ELSE	//Kasuje zeby po cyklu nic sie nie poruszało
	bManualCatchActuator := FALSE;
	bManualHeightMotorUp  := FALSE;
	bManualHeightMotorDown  := FALSE;
END_IF


IF bHoming OR bHeightSet THEN
	eState:=E_Station.eHoming;
END_IF
	
Running();
	
//Zabezpieczenie przed kolizją stacji poprzez ruch podnośnika	
IF bHeightMotorDown AND lrHeightMotorCV<=lrMinHeight AND NOT bHoming AND NOT bHeightSet THEN
	bHeightMotorDown:=FALSE;
END_IF	

IF bHeightMotorUp AND lrHeightMotorCV>=lrMaxHeight AND NOT bHoming AND NOT bHeightSet THEN
	bHeightMotorUp:=FALSE;
END_IF		 

IF NOT bRun THEN
	bCycleDone 					:= FALSE;
	bCycleNotDone 				:= FALSE;	
END_IF
END_ACTION

ACTION Running:

//Timery
tonCatchingTime(IN:=(eRunningState=E_CatchStationState.eCatching), PT:=T#500MS);


CASE eRunningState OF
	
	//NIEGOTOWY
	E_CatchStationState.eDisabled:
		eRunningState:=E_CatchStationState.eReady;

	//Chwytak gotowy do pracy
	E_CatchStationState.eReady: 
		//Jeśli komenda chwytania przejdz do stanu chwytanie
		IF NOT bCycleDone AND NOT bCycleNotDone THEN
			IF bRun THEN
			eRunningState:=E_CatchStationState.eCatching;
			END_IF
		END_IF
		
	//Chwytanie 
	E_CatchStationState.eCatching:
		bCatchActuator:=TRUE;
		

		IF tonCatchingTime.Q THEN
			IF bClosedActuatorSensor THEN
				eRunningState	:= E_CatchStationState.eCatched;
			ELSE
				eRunningState	:= E_CatchStationState.eNotCatched;
			END_IF
		END_IF

	//Uchwycone 
	E_CatchStationState.eCatched:
		bCatchActuator:=bRun;
		bCycleDone := TRUE;
		//Kiedy zniknie rozkaz chwytania i 
	
	E_CatchStationState.eNotCatched:
	
		bCatchActuator:=bRun;                                   
		bCycleDone := TRUE;
	
END_CASE
END_ACTION

ACTION Statistics:



rtrigCycleTimerRead(CLK:=eRunningState=E_CatchStationState.eCatched);
IF rtrigCycleTimerRead.Q THEN
	tCycleTime:=tonCycleTimer.ET;
END_IF
tonCycleTimer(IN:=eState>E_Station.eReady,PT:=T#1D);
END_ACTION

END_FUNCTION_BLOCK

// ---- POUs/FB/FB_FestoEmcsSt.TcPOU
FUNCTION_BLOCK FB_FestoEmcsSt
VAR_INPUT
	bEstop												:	BOOL;			//	FALSE = SAFETY
	//Control
	bHoming												:	BOOL;			//	Zbazować
	bSetIn												:	BOOL;  	 		//	Schowaj do końca
	bSetIntermidate										:	BOOL;  			//	Wysuń do pozycji intermidate
	bSetOut												:	BOOL;   		//	Wysuń do końca
	bMoveIn												:	BOOL;   		//	Ruch na schowanie (kasuje ruch po zdejmowaniu sygnału)  
	bMoveInter											:	BOOL;   		//	Ruch na pozycje intermidate (kasuje ruch po zdejmowaniu sygnału)
	bMoveOut											:	BOOL;   		//	Ruch na wysunęcie (kasuje ruch po zdejmowaniu sygnału)
	bPlsIn												:	BOOL;   		//	Krótki ruch (schowanie)
	bPlsOut												:	BOOL;   		//	Krótki ruch (wysunęcie)
	bReset												:	BOOL;   		//	Zresetuj błądy
	                                                                    	
	//FESTO DI                                                          	
	ibStateIn									AT%I* 	: 	BOOL;   		//	Festo: na pozycji SCHOWANY
	ibStateOut									AT%I* 	: 	BOOL;   		//  Festo: na pozycji WYSUNIĘTY
	ibStateDevice								AT%I* 	: 	BOOL;   		//  Festo: true => Device Ok, false - Bląd
	ibStateMove									AT%I* 	: 	BOOL;   		//  Festo: w trakcie ruchu
	ibStateIntermidate							AT%I* 	: 	BOOL;   		//  Festo: na pozycji INTERMIDATE
	
	bHomingDirectionInNotOut							:	BOOL; 			//	Kierunek bazowania	TRUE => Schowanie, FALSE => Wysunięcie
	
	tPlsLength											:	TIME:=T#40MS;	//	Czas krótkiego rucha
	
	sNetId												:	STRING 		:=''; //IoLink master Net Id 
	eIolPort											:	E_IolPort	;     //IoLinkPort
	
	rInterPos											:	REAL;	//Intermidate pozycja

	usiInSpeed											:	USINT;
	usiOutSpeed											:	USINT;
	usiForce											:	USINT;


END_VAR
VAR_OUTPUT
	eState												:	E_FestoEmcsStState;	//Status bloczka
	bHomingDone											:	BOOL;			//Flag homing done
	
	bError												:	BOOL;
	bBusy												:	BOOL;	
	bDone												:	BOOL;	
	//FESTO DO
	qbMoveIn									AT%Q* 	: 	BOOL;			//Festo: roskaz rusz na schowanie
	qbMoveOut									AT%Q* 	: 	BOOL;           //Festo: roskaz rusz na wysunięcie
	qbQuitError									AT%Q* 	: 	BOOL;           //Festo: roskaz resetuj błąd osi
	qbMoveIntermidate							AT%Q* 	: 	BOOL;           //Festo: roskaz rusz na intermidate
	
	udiErrorCode										:	UDINT;
END_VAR
VAR
	rtSetIn												:	R_TRIG;			//RTIG dla bSetIn
	rtSetIntermidate									:	R_TRIG;			//RTIG dla bSetInter
	rtSetOut											:	R_TRIG;			//RTIG dla bSetOut
	rtReset												:	R_TRIG;			//RTIG dla bReset
	rtPlsIn												:	R_TRIG;			//RTIG dla bPlsIn
	rtPlsOut											:	R_TRIG;			//RTIG dla bPlsOut
	tonLongActError										:	TON;			//Czasówka błędu 'Zbyt dluga operacja' 
	tonLongActError2									:	TON;			//Czasówka błędu 'Zbyt dluga operacja' 
	tonStatusControl									:	TON;			//Czasówka błędu od sterownika festo
	tonPls												:	TON;			//Czasówka dla krótkich ruchów
	tLongAct											:	TIME:=	T#25S;  //Czas kontroli blędu dlugej operacji (pierwszy homing 25s, kolejne operacje 5s)

	tonSafetyReset										:	TON;
	tonResetting										:	TON;
	

	(*ADS Io Operations*)
	
	//InterPosWrite
	udiInterPosWriteCase								:	UDINT;
	fbWrInterPos										:	FB_IolWrite;
	aWrInterPosTmp										:	ARRAY[0..3] OF BYTE;
	aWrInterPosTmpInv									:	ARRAY[0..3] OF BYTE;
	tonWrInterPosDone									:	ton;
	
	//In Out speeds & force
	fbWrInSpeed											:	FB_IolWrite;
	fbWrOutSpeed										:	FB_IolWrite;
	fbWrForce											:	FB_IolWrite;
	tonWrInSpeedDone									:	ton;
	tonWrOutSpeedDone									:	ton;
	tonWrForceDone										:	ton;

	//RefCmd
	fbWrRefMove											:	FB_IolWrite;
	bWrRefMove											:	BOOL	:=	TRUE;
	
	//Homing
	tonWaitRefWrite										:	TON;
	iHomingCase 										:	UDINT;

	usiInSpeedlast: USINT;
	usiOutSpeedLast: USINT;
END_VAR

ACT_Signals();
ACT_Control();
ACT_IoLinkViaAds();
ACT_ErrorHandling();

ACTION ACT_Control:
tonSafetyReset(IN:=bEstop,PT:=T#1S);
IF (NOT bEstop) THEN
	eState												:=	E_FestoEmcsStState.eEStop;
END_IF
	
IF (
	(	eState = E_FestoEmcsStState.eUnhomed 	OR
		eState = E_FestoEmcsStState.eUnknown 	OR
		eState = E_FestoEmcsStState.eIn			OR
		eState = E_FestoEmcsStState.eOut		OR
		eState = E_FestoEmcsStState.eInter		)   AND bHoming) THEN	
		bHomingDone										:=	FALSE;
		iHomingCase										:=	0;
		eState											:=	E_FestoEmcsStState.eHoming;
END_IF



CASE eState OF
	E_FestoEmcsStState.eEStop:
		ACT_EStop();
	
	E_FestoEmcsStState.eHoming:
		ACT_Homing();
		
	E_FestoEmcsStState.eHomingDone:
		ACT_HomingDone();

	E_FestoEmcsStState.eUnknown	,
	E_FestoEmcsStState.eIn		,
	E_FestoEmcsStState.eOut		,
	E_FestoEmcsStState.eInter		:
		ACT_OnPosition();

	E_FestoEmcsStState.ePlsIn,
	E_FestoEmcsStState.ePlsOut:
		ACT_Pls();
		
	E_FestoEmcsStState.eSettingIn:
		ACT_SetIn();
		
	E_FestoEmcsStState.eSettingOut:
		ACT_SetOut();
			
	E_FestoEmcsStState.eSettingInter:
		ACT_SetInter();
		
	E_FestoEmcsStState.eMoveIn:
		ACT_MoveIn();
		
	E_FestoEmcsStState.eMoveOut:
		ACT_MoveOut();
		
	E_FestoEmcsStState.eMoveInter:
		ACT_MoveInter();
				
	E_FestoEmcsStState.eError:
		ACT_Error();
		
	E_FestoEmcsStState.eResetting:
		ACT_Resetting();
		
END_CASE
END_ACTION

ACTION ACT_Error:
fbWrForce.bExecute										:=	FALSE;
fbWrInSpeed.bExecute									:=	FALSE;
fbWrOutSpeed.bExecute									:=	FALSE;
fbWrInterPos.bExecute									:=	FALSE;
fbWrRefMove.bExecute									:=	FALSE;
qbMoveIn												:=	FALSE;
qbMoveIntermidate										:=	FALSE;
qbMoveOut												:=	FALSE;
qbQuitError												:=	FALSE;
IF (rtReset.Q) THEN                             		
	eState												:=	E_FestoEmcsStState.eResetting;
END_IF
END_ACTION

ACTION ACT_ErrorHandling:
IF (tonLongActError.Q) THEN
	eState												:=	E_FestoEmcsStState.eError;
	udiErrorCode										:=	1000;
END_IF

tonStatusControl(IN:=NOT ibStateDevice, PT:=T#10S);

IF (tonLongActError2.Q) THEN
	eState												:=	E_FestoEmcsStState.eError;
	udiErrorCode										:=	2000;
END_IF

IF (
	tonStatusControl.Q						AND 
	eState <> E_FestoEmcsStState.eResetting AND 
	eState <> E_FestoEmcsStState.eEStop		AND 
	bHomingDone
	) THEN
	eState												:=	E_FestoEmcsStState.eError;
	CASE eState OF
		E_FestoEmcsStState.eUnhomed				:	udiErrorCode:=	5200;
		E_FestoEmcsStState.eHoming				:	udiErrorCode:=	5101;
		E_FestoEmcsStState.eHomingDone			:	udiErrorCode:=	5202;
		E_FestoEmcsStState.eUnknown				:	udiErrorCode:=	5203;
		E_FestoEmcsStState.eIn					:	udiErrorCode:=	5204;
		E_FestoEmcsStState.eOut					:	udiErrorCode:=	5205;
		E_FestoEmcsStState.eInter				:	udiErrorCode:=	5206;
		E_FestoEmcsStState.eMoveIn				:	udiErrorCode:=	5107;
		E_FestoEmcsStState.eSettingIn			:	udiErrorCode:=	5108;
		E_FestoEmcsStState.ePlsIn				:	udiErrorCode:=	5109;
		E_FestoEmcsStState.eMoveOut				:	udiErrorCode:=	5110;
		E_FestoEmcsStState.eSettingOut			:	udiErrorCode:=	5111;
		E_FestoEmcsStState.ePlsOut				:	udiErrorCode:=	5112;
		E_FestoEmcsStState.eMoveInter			:	udiErrorCode:=	5113;
		E_FestoEmcsStState.eSettingInter		:	udiErrorCode:=	5114;
		E_FestoEmcsStState.eError				:	udiErrorCode:=	5215;
		E_FestoEmcsStState.eResetting			:	udiErrorCode:=	5316;
		E_FestoEmcsStState.eEStop				:	udiErrorCode:=	5000;			
	END_CASE
END_IF
END_ACTION

ACTION ACT_EStop:
IF (tonSafetyReset.Q) THEN
	qbQuitError											:=	TRUE;
	IF (ibStateDevice) THEN
		qbQuitError										:=	FALSE;
		eState 											:= 	E_FestoEmcsStState.eUnknown; 
	END_IF
ELSE
	qbMoveIn											:=	FALSE;
	qbMoveIntermidate									:=	FALSE;
	qbMoveOut											:=	FALSE;
	qbQuitError											:=	FALSE;
END_IF
END_ACTION

ACTION ACT_Homing:
tonWaitRefWrite		(IN:= 	iHomingCase = 10,PT:=T#1S500MS);
tonWrInterPosDone	(IN:=	iHomingCase = 17,PT:=T#1500MS);
tonWrInSpeedDone	(IN:=	iHomingCase = 27,PT:=T#1500MS);
tonWrOutSpeedDone	(IN:=	iHomingCase = 37,PT:=T#1500MS);
tonWrForceDone		(IN:=	iHomingCase = 47,PT:=T#1500MS);

CASE iHomingCase OF
	0:
		bHomingDone										:=	FALSE;
		fbWrRefMove.bExecute							:=	TRUE;
		IF (fbWrRefMove.bDone) THEN
			fbWrRefMove.bExecute						:=	FALSE;
			iHomingCase									:=	10;
		END_IF
		IF (fbWrRefMove.bError) THEN
			eState										:=	E_FestoEmcsStState.eError;
			udiErrorCode								:=	3100;
			iHomingCase									:=	0;
		END_IF
	10:
		IF (tonWaitRefWrite.Q AND NOT ibStateMove AND ibStateOut) THEN
			//REAL kurwa w odwrotnej kolejnośći u Festo!!!!!
			Memcpy(ADR(aWrInterPosTmpInv),ADR(rInterPos),SIZEOF(aWrInterPosTmp));
			aWrInterPosTmp[0]:=aWrInterPosTmpInv[3];
			aWrInterPosTmp[1]:=aWrInterPosTmpInv[2];
			aWrInterPosTmp[2]:=aWrInterPosTmpInv[1];
			aWrInterPosTmp[3]:=aWrInterPosTmpInv[0];
			fbWrInterPos.bExecute						:=	TRUE;	
			iHomingCase									:=	15;
		END_IF                              		
	15:                                     		
		IF 	(fbWrInterPos.bError) THEN      		
			eState										:=	E_FestoEmcsStState.eError;
			udiErrorCode								:=	3200;
			iHomingCase									:=	0;
		END_IF                              		
		IF 	(fbWrInterPos.bDone) THEN       	
			fbWrInterPos.bExecute						:=	FALSE;	
			iHomingCase									:=	17;
		END_IF
	17:
		IF (tonWrInterPosDone.Q) THEN
			iHomingCase									:=	20;
		END_IF
	20:		
		IF (usiInSpeed<1 OR usiInSpeed>10) THEN
			usiInSpeed									:=	10;
		END_IF                                  		
		iHomingCase										:=	25;
		fbWrInSpeed.bExecute							:=	TRUE;
	25:                                         		
		IF 	(fbWrInSpeed.bError) THEN           		
			eState										:=	E_FestoEmcsStState.eError;
			udiErrorCode								:=	3200;
			iHomingCase									:=	0;
		END_IF                                  		
		IF 	(fbWrInSpeed.bDone) THEN            		
			fbWrInSpeed.bExecute						:=	FALSE;	
			iHomingCase									:=	27;
		END_IF                                  	
	27:                                         	
		IF (tonWrInSpeedDone.Q) THEN            	
			iHomingCase									:=	30;
		END_IF
	30:		
		IF (usiOutSpeed<1 OR usiOutSpeed>10) THEN
			usiOutSpeed									:=	10;
		END_IF                                  		
		iHomingCase										:=	35;
		fbWrOutSpeed.bExecute							:=	TRUE;
	35:                                         		
		IF 	(fbWrOutSpeed.bError) THEN          		
			eState										:=	E_FestoEmcsStState.eError;
			udiErrorCode								:=	3400;
			iHomingCase									:=	0;
		END_IF                                  		
		IF 	(fbWrOutSpeed.bDone) THEN           		
			fbWrOutSpeed.bExecute						:=	FALSE;	
			iHomingCase									:=	37;
		END_IF                                  		
	37:                                         		
		IF (tonWrOutSpeedDone.Q) THEN           		
			iHomingCase									:=	40;
		END_IF                                  		
	40:		                                    		
		IF (usiForce<1 OR usiForce>10) THEN     		
			usiForce									:=	1;
		END_IF                                  		
		iHomingCase										:=	45;
		fbWrForce.bExecute								:=	TRUE;
	45:                                         		
		IF 	(fbWrForce.bError) THEN             		
			eState										:=	E_FestoEmcsStState.eError;
			udiErrorCode								:=	3500;
			iHomingCase									:=	0;
		END_IF                                  		
		IF 	(fbWrForce.bDone) THEN              		
			fbWrForce.bExecute							:=	FALSE;	
			iHomingCase									:=	47;
		END_IF	                                		
	47:                                         		
		IF (tonWrForceDone.Q) THEN              		
			iHomingCase									:=	50;
		END_IF                                  		
	50:    
		usiInSpeedLast									:=  usiInSpeed;	
		usiOutSpeedLast									:=  usiOutSpeed;		                                   		
		bHomingDone										:=	TRUE;
		iHomingCase										:=	0;
		eState											:=	E_FestoEmcsStState.eHomingDone;
END_CASE
END_ACTION

ACTION ACT_HomingDone:
IF (NOT bHoming) THEN
	eState												:=	E_FestoEmcsStState.eUnknown;
END_IF
END_ACTION

ACTION ACT_IoLinkViaAds:
//Reference movement
fbWrRefMove.cbBufLen		:=	SIZEOF(bWrRefMove);
fbWrRefMove.nIndex			:=	16#0104;
fbWrRefMove.nIolPort		:=	eIolPort;
fbWrRefMove.nSubindex		:=	16#0000;
fbWrRefMove.pSRCBuf			:=	ADR(bWrRefMove);
fbWrRefMove.sNetId			:=	sNetId;
fbWrRefMove.tTimeout		:=	T#2S;
fbWrRefMove();


//InterPosWrite
fbWrInterPos.cbBufLen		:=	SIZEOF(aWrInterPosTmp);
fbWrInterPos.nIndex			:=	16#0108;
fbWrInterPos.nIolPort		:=	eIolPort;
fbWrInterPos.nSubindex		:=	16#0000;
fbWrInterPos.pSRCBuf		:=	ADR(aWrInterPosTmp);
fbWrInterPos.sNetId			:=	sNetId;
fbWrInterPos.tTimeout		:=	T#2S;
fbWrInterPos();

//InSpeed
fbWrInSpeed.cbBufLen		:=	SIZEOF(usiInSpeed);
fbWrInSpeed.nIndex			:=	16#0100;
fbWrInSpeed.nIolPort		:=	eIolPort;
fbWrInSpeed.nSubindex		:=	16#0000;
fbWrInSpeed.pSRCBuf			:=	ADR(usiInSpeed);
fbWrInSpeed.sNetId			:=	sNetId;
fbWrInSpeed.tTimeout		:=	T#2S;
fbWrInSpeed();

//OutSpeed
fbWrOutSpeed.cbBufLen		:=	SIZEOF(usiOutSpeed);
fbWrOutSpeed.nIndex			:=	16#0101;
fbWrOutSpeed.nIolPort		:=	eIolPort;
fbWrOutSpeed.nSubIndex		:=	16#0000;
fbWrOutSpeed.pSRCBuf		:=	ADR(usiOutSpeed);
fbWrOutSpeed.sNetId			:=	sNetId;
fbWrOutSpeed.tTimeout		:=	T#2S;
fbWrOutSpeed();

//Force
fbWrForce.cbBufLen			:=	SIZEOF(usiForce);
fbWrForce.nIndex			:=	16#0102;
fbWrForce.nIolPort			:=	eIolPort;
fbWrForce.nSubindex			:=	16#0000;
fbWrForce.pSRCBuf			:=	ADR(usiForce);
fbWrForce.sNetId			:=	sNetId;
fbWrForce.tTimeout			:=	T#2S;
fbWrForce();

IF usiInSpeedLast <>	usiInSpeed AND bHomingDone THEN
	fbWrInSpeed.bExecute		:= TRUE;
	IF fbWrInSpeed.bDone OR fbWrInSpeed.bError THEN
		fbWrInSpeed.bExecute	:=  FALSE;
	END_IF
	IF fbWrInSpeed.bDone THEN
		usiInSpeedLast			:=	usiInSpeed;
	END_IF	
END_IF

IF usiOutSpeedLast <>	usiOutSpeed AND bHomingDone THEN
	fbWrOutSpeed.bExecute		:= TRUE;
	IF fbWrOutSpeed.bDone OR fbWrOutSpeed.bError THEN
		fbWrOutSpeed.bExecute	:=  FALSE;
	END_IF
	IF fbWrOutSpeed.bDone THEN
		usiOutSpeedLast			:=	usiOutSpeed;
	END_IF	
END_IF
END_ACTION

ACTION ACT_MoveIn:
IF (ibStateIn OR NOT bMoveIn) THEN
	qbMoveIn											:=	FALSE;
	eState												:=	E_FestoEmcsStState.eUnknown;
END_IF
END_ACTION

ACTION ACT_MoveInter:
IF (ibStateIntermidate OR NOT bMoveInter) THEN
	qbMoveIntermidate									:=	FALSE;
	eState												:=	E_FestoEmcsStState.eUnknown;
END_IF
END_ACTION

ACTION ACT_MoveOut:
IF (ibStateOut OR NOT bMoveOut) THEN
	qbMoveOut											:=	FALSE;
	eState												:=	E_FestoEmcsStState.eUnknown;
END_IF
END_ACTION

ACTION ACT_OnPosition:
qbMoveIn										:=	FALSE;
qbMoveIntermidate								:=	FALSE;
qbMoveOut										:=	FALSE;
IF (ibStateIn) THEN
	eState										:=	E_FestoEmcsStState.eIn;
ELSIF (ibStateOut) THEN
	eState												:=	E_FestoEmcsStState.eOut;
ELSIF (ibStateIntermidate) THEN
	eState												:=	E_FestoEmcsStState.eInter;
END_IF
		
IF (rtSetIn.Q AND NOT ibStateIn) THEN
	qbMoveIn											:=	TRUE;
	eState												:=	E_FestoEmcsStState.eSettingIn;
ELSIF (rtSetOut.Q AND NOT ibStateOut) THEN
	qbMoveOut											:=	TRUE;
	eState												:=	E_FestoEmcsStState.eSettingOut;
ELSIF (rtSetIntermidate.Q AND NOT ibStateIntermidate) THEN
	qbMoveIntermidate									:=	TRUE;
	eState												:=	E_FestoEmcsStState.eSettingInter;
ELSIF (bMoveIn AND NOT ibStateIn) THEN
	qbMoveIn											:=	TRUE;
	eState												:=	E_FestoEmcsStState.eMoveIn;
ELSIF (bMoveOut AND NOT ibStateOut) THEN
	qbMoveOut											:=	TRUE;
	eState												:=	E_FestoEmcsStState.eMoveOut;
ELSIF (bMoveInter AND NOT ibStateIntermidate) THEN
	qbMoveIntermidate									:=	TRUE;
	eState												:=	E_FestoEmcsStState.eMoveInter;
ELSIF (rtPlsIn.Q AND NOT ibStateIn) THEN
	qbMoveIn											:=	TRUE;
	eState												:=	E_FestoEmcsStState.ePlsIn;
ELSIF (rtPlsOut.Q AND NOT ibStateOut) THEN
	qbMoveOut											:=	TRUE;
	eState												:=	E_FestoEmcsStState.ePlsOut;		
END_IF
END_ACTION

ACTION ACT_Pls:
IF (tonPls.Q) THEN
	bDone												:=	TRUE;
	qbMoveIn											:=	FALSE;
	qbMoveOut											:=	FALSE;
	eState												:=	E_FestoEmcsStState.eUnknown;
END_IF
END_ACTION

ACTION ACT_Resetting:
qbQuitError												:=	TRUE;
IF (ibStateDevice AND tonResetting.Q) THEN
	bDone												:=	TRUE;
	udiErrorCode										:=	0;
	qbQuitError											:=	FALSE;
	eState												:=	E_FestoEmcsStState.eUnknown;
END_IF
END_ACTION

ACTION ACT_SetIn:
IF (ibStateIn) THEN
	bDone												:=	TRUE;
	qbMoveIn											:=	FALSE;
	eState												:=	E_FestoEmcsStState.eIn;
END_IF
END_ACTION

ACTION ACT_SetInter:
IF (ibStateIntermidate) THEN
	bDone												:=	TRUE;
	qbMoveIntermidate									:=	FALSE;
	eState												:=	E_FestoEmcsStState.eInter;
END_IF
END_ACTION

ACTION ACT_SetOut:
IF (ibStateOut) THEN
	bDone												:=	TRUE;
	qbMoveOut											:=	FALSE;
	eState												:=	E_FestoEmcsStState.eOut;
END_IF
END_ACTION

ACTION ACT_Signals:
rtSetIn				(CLK:=	bSetIn				);
rtSetIntermidate	(CLK:=	bSetIntermidate		);
rtSetOut			(CLK:=	bSetOut				);
rtReset				(CLK:=	bReset				);
rtPlsIn				(CLK:=	bPlsIn				);
rtPlsOut			(CLK:=	bPlsOut				);

tonResetting(IN:=qbQuitError, PT:=T#500MS);

tonPls(IN:= (eState = E_FestoEmcsStState.ePlsIn OR eState = E_FestoEmcsStState.ePlsOut),PT:=tPlsLength);

bBusy													:=
	eState	=	E_FestoEmcsStState.eMoveIn 			OR
	eState	=	E_FestoEmcsStState.eMoveInter 		OR
	eState	=	E_FestoEmcsStState.eMoveOut 		OR
	eState	=	E_FestoEmcsStState.eSettingIn 		OR
	eState	=	E_FestoEmcsStState.eSettingInter 	OR
	eState	=	E_FestoEmcsStState.eSettingOut 		OR
	eState	=	E_FestoEmcsStState.eResetting		OR
	eState	=	E_FestoEmcsStState.eHoming;

tonLongActError (IN:= bBusy AND eState	<>	E_FestoEmcsStState.eHoming , PT:=tLongAct);
tonLongActError2(IN:= bBusy AND eState	=	E_FestoEmcsStState.eHoming , PT:=T#60S);

bError													:=	eState = E_FestoEmcsStState.eError;	

IF (NOT (bSetIn OR bSetIntermidate OR bSetOut OR bReset OR bPlsIn OR bPlsOut)) THEN
	bDone												:=	FALSE;
END_IF
END_ACTION

END_FUNCTION_BLOCK

// ---- POUs/FB/FB_SensorDiag.TcPOU
(*
Nazwa:			FB_SensorDiag
Opis: 			Diagnostyka czujników
Wersja:			v0.1
Data:			2024-05-27
Autor:			DP
Urzadzenia:		
Konfiguracja:	
Info:
- Diagnostyka czujnika
*)

FUNCTION_BLOCK FB_SensorDiag
VAR_INPUT
	bSensor					:BOOL;			// Wejście czujnika
	bReset					:BOOL;
	sSensorName				:STRING(200);	// Nazwa
	bShouldBlinking			:BOOL;
	tTimeToError			:TIME;			// Czas do błędu
	
	iStationIndex			:UDINT;			// Numer stacji 
	sStationName			:STRING;		// Nazwa stacji
END_VAR
VAR_OUTPUT
	bError					:BOOL;
	udiErrorID				:UDINT;	
	sErrorStationName		:STRING;							
	sErrorDescription		:STRING(200);
	sErrorDescription2		:STRING(200);	
END_VAR
VAR
	tonNoBlinkingAndOn		:TON;
	tonNoBlinkingAndOff		:TON;	
END_VAR


tonNoBlinkingAndOff	(IN:= bShouldBlinking AND NOT bSensor,	PT:=tTimeToError);
tonNoBlinkingAndOn	(IN:= bShouldBlinking AND bSensor, 		PT:=tTimeToError);
	
IF (tonNoBlinkingAndOff.Q OR tonNoBlinkingAndOn.Q) AND NOT bError THEN
	bError					:=	TRUE;
	IF tonNoBlinkingAndOff.Q THEN
		udiErrorID			:= 	1	+	iStationIndex;	
		sErrorDescription	:=	' Błąd czujnika - ciągły sygnał "0"'; 
	ELSIF tonNoBlinkingAndOn.Q THEN
		udiErrorID			:= 	2	+	iStationIndex;					
		sErrorDescription	:=	' Błąd czujnika - ciągły sygnał "1"'; 
	END_IF	
END_IF

IF bReset THEN
	bError					:=	FALSE;
END_IF

sErrorDescription2			:= sSensorName;
sErrorStationName			:= sStationName;

END_FUNCTION_BLOCK

// ---- POUs/FB/FB_ServoDispencerServoLifter_kopia_przed_akt_XTS.TcPOU
(*
Nazwa:			FB_ServoDispencerFestoLifter
Opis:			Dozownik 
Wersja:			v0.5
Data:			2019-07-31
Autor:			DP
Urzadzenia:		Serwo dozowania, silniki krokowe podnoszenia FESTO, zawor ssania-dozowania
Konfiguracja:	
Info: 
-Zmieniono zachowanie po HomingDone
-Dodano opisy błędów serwa
-Zmiana zachowania tacki po wylaczeniu enable
-Dodano HomingNeeded
-Ulepszono przerywanie dozowania
-Enable Festo, dopiero jak nie ma warningu i jest zasilanie
-falsowanie enable festo na koncu
-Dodanie wysokosci tacki okapowej
*)
FUNCTION_BLOCK FB_ServoDispencerServoLifter_kopia_przed_akt_XTS
VAR_INPUT
    bEnable              : BOOL;          //Zezwolenie na pracę
	bChangover 				:BOOL;	
    bEStop               : BOOL;          //Stop Awaryjny Całość
    bEStopButtonsAndDoors: BOOL;          //Stop Awaryjny	
	bInLimitSwitchSensor : BOOL; 		  //Krańcówka dosunięcia stacji
    bRun                 : BOOL;          //Rozkaz dozowania 
    bHoming              : BOOL;          //Zezwolenie na wykonanie bazowania (głównie po wykonanych mechanicznych zmianach)
    bHeightSet           : BOOL;          //Zezwolenie na wykonanie bazowania (głównie po wykonanych mechanicznych zmianach)
    bIgnoreError         : BOOL;          //Ignorowania błędów cyklu pracy
    bReset               : BOOL;          //Reset błędu, jeśli w stanie "eError"
    eGlobalState         : E_PackMLState; //Stan ogólny maszyny, tylko do błędu
    bCatchEnable         : BOOL;          //Zezwolenie na pracę chwytaka, tylko do błędu
    lrDoseVolume         : LREAL;         //Ilość do wydozowania w [ml]
    bDispencerWithLifter : BOOL;          //OPCJA Dozownik z podnośnikiem
    bMultiMasterSyncIn   : BOOL;          //OPCJA Synchronizacja gotowsci innych dozowników // Jezeli ma działać niezależnie to ma być cały czas na TRUE
    bLiftSynchroPh1      : BOOL;          //Synchronizacja podnośnika z Dozownikiem w fazie 1
    bLiftSynchroPh2      : BOOL;          //Synchronizacha podnośnika z Dozownikiem w fazie 2
    bLiftSynchroPh3      : BOOL;          //Synchronizacja podnośnika z Dozownikiem w fazie 3

    //Parametryzacja dozownika (można wpisać na stałe)
    lrMaxPosition      			: LREAL; 		//Pozycja maksymalna podnośnika
    lrMinPosition      			: LREAL; 		//Pozycja minimalna podnośnika
    lrRatedDose        			: LREAL; 		//Znamionowa pojemność dozownika [ml];
    lrCylinderDiameter 			: LREAL;		//Średnica cylindra dozownika [mm]
	lrDropCatcherOpenDistance	: LREAL:=10;	//Różnica od aktualnej wysokości chwytaka przy której ma się otworzyć tacka (Domyślnie 10)
	
    //Informacje z czujników
    bSuckingValveOpenedSensor : BOOL;  //Czujnik otwarcia zaworu ssacego
    bSuckingValveClosedSensor : BOOL;  //Czujnik zamkmnięcia zaworu ssącego
    bDosingValveOpenedSensor  : BOOL;  //Czujnik otwarcia zaworu tłoczącego (iglicy)
    bDosingValveClosedSensor  : BOOL;  //Czujnik zamknięcia zaworu tłoczącego (iglicy) (tylko ten ma znaczenie w cyklu)
    bDropCatcherBackSensor    : BOOL;  //Czujnik wycofania tacki kropel
    lrLifterPullingPosition   : LREAL; //Pozycja podnośnika podczas przeciągania (podpinaj jeśli bDispencerWithLifter, innaczej pozostaw bez zmiennej)

    //WEJSCIA WYJSCIA SPRZETOWE
    // DO FML_READ
    // Struktura osi
    lrDropCatcherHeightCV : LREAL; // Aktualna wysokość tacki okapowej

    //WEJSCIA WYJSCIA SPRZETOWE
    iStationIndex : UDINT;  //Numer stacji 
    sStationName  : STRING; //Nazwa stacji
END_VAR
VAR_OUTPUT
    eState                 : E_Station;        //Stan ogólny bloku	
    eRunningState          : E_DispencerState; //Stan dozownika
    bError                 : BOOL;             //Błąd stacji
    nErrorNr               : UDINT;            //Nr błędu dozownika
    sErrorDescription      : STRING(200);      //Opis błędu
    sErrorDescription2     : STRING(200);      //Opis błędu
    sErrorStationName      : STRING;           //Nazwa stacji	
    nDispencerServoErrorNr : UDINT;            //Nr błędu serwo nalewarki
    nLifterServoErrorNr    : UDINT;            //Nr błędu serwo podnośnika
    lrDosedMassCV          : LREAL;            //Aktualna wydozowana doza
    bSuckingValveActuator  : BOOL;             //Siłownik zaworu ssącego
    bDosingValveActuator   : BOOL;             //Siłownik Zaworu tłoczącego
    bDropCatcherActuator   : BOOL;             //Siłownik tacki kropel	
    tCycleTime             : TIME;
    bCyclePrepareDone      : BOOL;
    bCycleDone             : BOOL;
    bCycleNotDone          : BOOL;
    bDosingDoneDelayOutput : BOOL;

    lrLifterActualPosition : LREAL; // Aktualna pozycja podnosnika dozownika
    bEncoderHomed          : BOOL;  // Dozowniki zbazowane
    bHomingDone            : BOOL;  //Wymagane ponowne bazowanie (blad podczas bazowania lub stop awaryjny)
    bMultiMasterSyncOut    : BOOL;  //OPCJA Synchronizacja gotości dozownika
END_VAR
VAR_IN_OUT

    //Fazy dozownika przy dozowaniu i ssaniu - jeśli wartości równe 0 faza zostanie pominięta. Następujące fazy muszą być od siebie większe	
    lrDosePhase1Volume        : LREAL; //Faza 1 dozowania (Podnośnik nieruchomy), do jakiej objętości ma trwać w [ml], następnie zaczyna sie 2 faza (powinna być mniejsza niż zadana objętość)
    lrDosePhase2Volume        : LREAL; //Faza 2 dozowania (Podnośnik zsynchronizowany z dozownikiem), do jakiej objętości ma trwać w [ml], następnie zaczyna sie 3 faza (powinna być mniejsza niż zadana objętość dozowania i większa od fazy 1)
    lrDosePhase1Velocity      : LREAL; //Prędkość dozowania Fazy 1 [ml/s]
    lrDosePhase2Velocity      : LREAL; //Prędkość dozowania Fazy 2 [ml/s] 
    lrDosePhase3Velocity      : LREAL; //Prędkość dozowania Fazy 3 [ml/s] 
    lrSuckVelocity            : LREAL; //Prędkość zasysania [ml/s] 
    lrDosePhase1Acceleration  : LREAL; //Przyspieszenie dozowania Fazy 1 [ml/s2]
    lrDosePhase2Acceleration  : LREAL; //Przyspieszenie dozowania Fazy 2 [ml/s2] 
    lrDosePhase3Acceleration  : LREAL; //Przyspieszenie dozowania Fazy 3 [ml/s2] 
    lrSuckAcceleration        : LREAL; //Przyspieszenie zasysania [ml/s2] 
    lrDosePhase1Deceleration  : LREAL; //Zwalnianie dozowania Fazy 1 [ml/s2]
    lrDosePhase2Deceleration  : LREAL; //Zwalnianie dozowania Fazy 2 [ml/s2] 
    lrDosePhase3Deceleration  : LREAL; //Zwalnianie dozowania Fazy 3 [ml/s2] 
    nDosingDoneDelayTime      : UDINT; //Czas odpóźnienia wykonania dozy [ms]
    lrSuckDeceleration        : LREAL; //Zwalnianie zasysania [ml/s2] 
    lrSuckValveOpenVolume     : LREAL; //Otwarcie zaworu ssącego po zadanej odległości od początku ssania [ml]
    lrSuckValveCloseVolume    : LREAL; //Zamknięcie zaworu ssącego po zadanej odległości od końca ssania [ml]
    lrDosingValveOpenVolume   : LREAL; //Otwarcie zaworu tłoczącego po zadanej odległości od początku tłoczenia [ml]
    lrDosingValveCloseVolume  : LREAL; //Zamknięcie zaworu tłoczącego po zadanej odległości od końca tłoczenia [ml]
    lrLifterReadyPosition     : LREAL; //Pozycja podnośnika dozownika przy starcie dozowania (podpinaj jeśli bDispencerWithLifter, innaczej pozostaw bez zmiennej)
    lrLifterStartDosePosition : LREAL; //Pozycja podnośnika dozownika przy starcie dozowania (podpinaj jeśli bDispencerWithLifter, innaczej pozostaw bez zmiennej)
    lrLifterStopDosePosition  : LREAL; //Pozycja podnośnika dozownika przy starcie dozowania (podpinaj jeśli bDispencerWithLifter, innaczej pozostaw bez zmiennej)
    lrLifterVelocity          : LREAL; //Prędkość podnosnika dozownika (podpinaj jeśli bDispencerWithLifter, innaczej pozostaw bez zmiennej)
    lrLifterAcceleration      : LREAL; //Przyspieszenie podnośnika dozownika(podpinaj jeśli bDispencerWithLifter, innaczej pozostaw bez zmiennej)
    lrLifterDeceleration      : LREAL; //Zwalnianie podnośnika dozownika  (podpinaj jeśli bDispencerWithLifter, innaczej pozostaw bez zmiennej)
  

    lrSuckValveOpenTimeDelay  : LREAL := 0; (*NOWA 0-1000*) // [3] Opóżnienie rozpoczęcia ssania po tłoczeniu [ms]
    lrSuckValveCloseTimeDelay : LREAL := 0; (*NOWA 0-2000*) // [4] Opóżnienie zamknięcia zaworu ssącego [ms]
    lrDoseValveOpenTimeAcc    : LREAL := 0; (*NOWA 0-500*)  // [1] Przyśpieszenie otwarcia zaworu tłoczenia [ms]
    lrDoseValveCloseTimeDec   : LREAL := 0; (*NOWA 0-1000*) // [2] Opóźnienie zamknięcia zaworu tłoczenia [ms]
    lrDoseSuckingVolume       : LREAL := 0; (*NOWA 0-100*)  // [5] [Podsysanie] Wartość dozy do posysenia [ml]	
    lrDoseSuckingTimeDelay    : LREAL := 0; (*NOWA 0-500*)  // [6] [Podsysanie] Opóźnienie podsysania [ms]
    bDoseSucking              : BOOL; (*NOWA*)              // [Podsysanie] Opcja podsysania przy dozowaniu

    //Ruchy ręczne
    bManualMovement           : BOOL;  //Zezwolenie na ruchy ręczne
    lrManualOverride          : LREAL; //Procentowa redukcja prędkości wszystkich serw (Tylko w trybie serwisowym)
    bManualPullingFast        : BOOL;  //Przeciąganie dozownika szybkie
    bManualPullingSlow        : BOOL;  //Przeciąganie dozownika wolne
	bManualCleaningMode		  : BOOL;	//Włączenie trybu mycia
	bManualCleaning			  : BOOL;	//Włącz mycie, do synchronizacji
    bManualPistonBack         : BOOL;  //Ruch ręczny podnośnikiem stacji w górę
    bManualPistonForward      : BOOL;  //Ruch ręczny podnośnikiem stacji w dół
    bManualSuckingValve       : BOOL;  //Otwarcie ręczne zaworu ssącego
    bManualDosingValve        : BOOL;  //Otwarcie ręczne zaworu dozującego (iglicy)
    bManualDropCatcherForward : BOOL;  //Wysunięcie ręczne tacki kropel
    bManualLifterUp           : BOOL;  //Podniesienie ręczne stacji dozownika (podpinać zmienną jeśli bDispencerWithLifter=TRUE)
    bManualLifterDown         : BOOL;  //Opuszczenie ręczne stacji dozownika (podpinać zmienną jeśli bDispencerWithLifter=TRUE)

    //Struktury NC
    DispencerAxisRef       : AXIS_REF; //Struktura sterowania NC dla serwa Dozownika
    DispencerLifterAxisRef : AXIS_REF;
    //Hamulec
    bServiceBrakeOff : BOOL; //Wyłączenie serwisowe hamulca  

END_VAR
VAR
    mcDispencerMoveAbsolute1 : MC_MoveAbsolute; // Blok nr 1 ruchu absolutnego tłoka dozownika
    mcDispencerMoveAbsolute2 : MC_MoveAbsolute; // Blok nr 2 ruchu absolutnego tłoka dozownika
    mcDispencerManualMove    : MC_JOG;          // Blok ruchu manualnego tłokiem dozownika
    mcDispencerStop          : MC_Stop;         // Blok zatrzymania tłoka dozownika, jeśli to konieczne
    mcDispencerSoftReset     : MC_Reset;        // Blok łagodnego resetu serwa tloka dozownika
    mcDispencerPower         : Mc_Power;        // Blok zasilania serwa dozownika
    bDispencerServoPower     : BOOL;            // Zalaczenie zasilania serwa
    // Blok resetowania twardego błędu
    fbDispencerHardReset : FB_SoEReset;
    // Blok Resetowania twardego błędu podnośnika

    // Pozycja przy rozpoczeciu dozowania
    lrStartDosingPos : LREAL;
    // Pozycja startowa tłoka dozownika przy rozpoczęciu zasysania
    lrSuckingMassStart : LREAL;
    // Ruch absolutny fazy 3
    mcDispencerMoveAbsolute3 : MC_MoveAbsolute;
    tonCycleTimer            : TON;
    rtrigCycleTimerRead      : R_TRIG;
    // zablokowanie przeciągania
    bManualPullingLatch : BOOL;
    // Opóźnienie przejścia do stanu zakończenia dozowania
    tonDosingDoneDelay : TON;
    bStopped           : BOOL;

    tonSuckingValveCloseError : TON; // Błąd zamknięcia zaworu ssącego
    tonSuckingValveOpenError  : TON; // Błąd otwarcia zaworu ssącego
    tonDosingValveCloseError  : TON; // Błąd zamknięcia zaworu dozującego
    tonDosingValveOpenError   : TON; // Błąd otwarcia zaworu dozującego

    tonSuckValveOpenTimeDelay  : TON;
    tonSuckValveCloseTimeDelay : TON;
    tonDoseValveOpenTimeAcc    : TON;
    tonDoseValveCloseTimeDec   : TON;
    tonDoseSuckingTimeDelay    : TON;

    (**********FESTO PODNOŚNIK ******************)
    // Blok Resetowania twardego błędu podnośnika
    fbLifterHardReset : FB_SoEReset;
    // Blok miekkiego resetu serwa podnosnika
    mcLifterSoftReset : MC_Reset;
    // Blok ruchu absolutnego podnosnika
    mcLifterMoveAbsolute : MC_MoveAbsolute;
    // Blok ruchu manualnego podnosnika
    mcLifterManualMove : MC_JOG;
    // Blok stopu podnosnika
    mcLifterStop : MC_Stop;
    // Blok zasilania serwa podnosnika
    mcLifterPower : Mc_Power;
    // Blok sprzęgania Dozownka z podnoszeniem
    mcLifterGearIn : Mc_GearInDyn;
    // Współczynnika przkeładni przy sprzeganiu dozownika z podnosnikiem (Wyliczany)
    lrGearRatio : LREAL;
    // Blok wysprzeglania dozownika i podnosnika
    mcLifterGearOut : Mc_GearOut;
    // Zasilanie serwo podnośnika dozownika
    bLifterServoPower     : BOOL;
    mcLifterGearInEnable  : BOOL;
    tofReset              : TOF;
	tonEstopDelay		  : TON;
    tonReadErrroFesto     : TON;
    rtLiftSynchroPh3      : R_TRIG;
    rtLiftSynchroPh2      : R_TRIG;
    rtLiftSynchroPh1      : R_TRIG;
    bPrepareToAborting    : BOOL;
    tonPrepareToAborting  : TON;
    lrPullingVelocity     : LREAL;
    TimerLifterNotEnabled : TON;
    rtDosingPh1           : R_TRIG;
    rtDosingPh2           : R_TRIG;
    rtDosingPh3           : R_TRIG;
    rtGoingUp             : R_TRIG;
    rtPreparingToDose     : R_TRIG;

    //Zabezpieczenie niektórych błędów aby pojawiały się tylko w cyklu
    bErrorOnlyIfCycleOn     : BOOL;
    tonDropCatcherOpenError : TON;
    tonStartHoming          : TON;
    lrLifterMaxHeight       : LREAL;
    lrLifterMinHeight       : LREAL;
    nCountCheckDisp1        : INT;
    nCheckCount123          : INT;
    nCheckCount124          : INT;
    nCheckCount125          : INT;
    ninttest                : INT;
    tonTooLongDosing        : TON;
    nCheckCount1233         : INT;
    nCheckCount1234         : INT;
    nCheckCount1235         : INT;
    nCheckCount1263         : INT;
    nCheckCount1236         : INT;
    tonEror10LifterNotReady : TON;
    nCountErr9              : INT;
    tonEror9LifterNotReady  : TON;
    bStateError             : BOOL;
    eLastState              : E_Station;        //Stan ogólny bloku
    eLastRunningState       : E_DispencerState; //Stan podbloku
    eLastStateTemp          : E_Station;        //Stan ogólny bloku
    eLastRunningStateTemp   : E_DispencerState; //Stan podbloku
    bPreparingToDisable     : BOOL;
    btestgoingup            : INT;
    bCountTestDoz1          : INT;
    bCountTestDoz2          : INT;

    bHeightSetNotDone : BOOL;

    mcHeightManualMove : INT;
    nCountTest12       : INT;
    bTest              : BOOL;
    trzeciafaza        : LREAL;
    drugafaza          : LREAL;
    calosc             : LREAL;
    tonDelayServoOn    : TON;
	tonDelayEnable: TON;
	
	//Bazowanie 
	bHardwareHoming				: BOOL;
	mcHardwareHomingPower		: MC_Power;
	fbHardwareHoming			: FB_HomingTorque;	

END_VAR

IF NOT bHardwareHoming THEN
	ErrorHandling();
	Control();
	Limits();
	DispencerControlBlocks();
	
	IF bDispencerWithLifter THEN 
		LifterControlBlocks();	
	END_IF
ELSE
	HardwareHoming();
	DispencerAxisRef();
	DispencerAxisRef.NcToPlc.ActTorque;
	DispencerAxisRef.NcToPlc.ActPos;
	DispencerAxisRef.Status.Homed;
END_IF
AntyColision();
Statistics();



(*wypracowanie sygnałów wyjściowych z bloku*)
lrLifterActualPosition:=DispencerLifterAxisRef.NcToPlc.ActPos; 	//Pozycja 
//bHomingDone:=Lifter_FHPP_CTRL.HomingValid; DP

(*Przepisywanie aktualnie wydozowanej ilości do butelki*)
//1,2,3 faza
IF eRunningState>6 AND eRunningState<11 THEN
	lrDosedMassCV:=DispencerAxisRef.NcToPlc.ActPos-lrDoseVolume;
ELSE
	lrDosedMassCV:=0;
END_IF
(*Koniec przepisywanie aktualnie wydozowanej ilości do butelki*)

(*Zapisywanie ostatniego stanu*)
IF eLastStateTemp<>eState THEN
	eLastState := eLastStateTemp;
END_IF
eLastStateTemp := eState;
IF eLastRunningStateTemp<>eRunningState THEN
	eLastRunningState := eLastRunningStateTemp;
END_IF
eLastRunningStateTemp := eRunningState;
(*Koniec Zapisywanie ostatniego stanu*)

ACTION AntyColision:
(*Zabezpieczenie przed kolizją stacji poprzez ruch podnośnika*)	
IF bManualLifterDown AND DispencerLifterAxisRef.NcToPlc.ActPos<=lrMinPosition AND NOT bHoming AND NOT bHeightSet THEN
	bManualLifterDown:=FALSE;
END_IF	

IF bManualLifterUp AND DispencerLifterAxisRef.NcToPlc.ActPos>=lrMaxPosition AND NOT bHoming AND NOT bHeightSet THEN
	bManualLifterUp:=FALSE;
END_IF
END_ACTION

